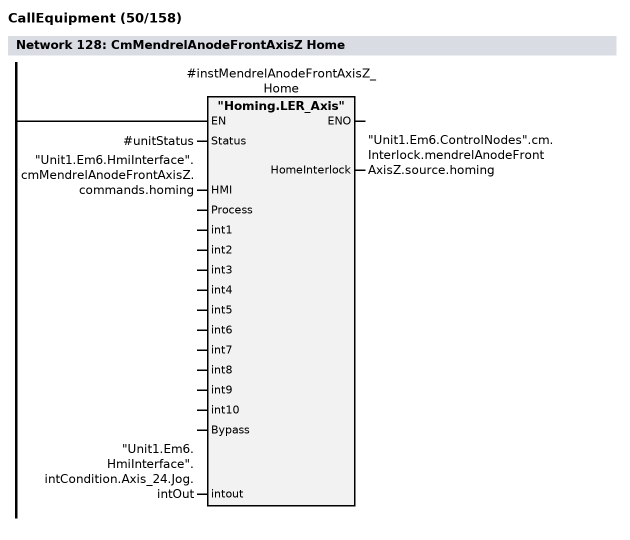
   RUNG wire#powerrail
      #instMendrelAnodeFrontAxisZ_Home(Status := #unitStatus, HMI := "Unit1.Em6.HmiInterface".cmMendrelAnodeFrontAxisZ.commands.homing, Process :=, int1 :=, int2 :=, int3 :=, int4 :=, int5 :=, int6 :=, int7 :=, int8 :=, int9 :=, int10 :=, Bypass :=, intout := "Unit1.Em6.HmiInterface".intCondition.Axis_24.Jog.intOut, HomeInterlock => "Unit1.Em6.ControlNodes".cm.Interlock.mendrelAnodeFrontAxisZ.source.homing)
   END_RUNG
   // the same network as SCL:
   #instMendrelAnodeFrontAxisZ_Home(Status := #unitStatus,   // "Homing.LER_Axis"
                           HMI := "Unit1.Em6.HmiInterface".cmMendrelAnodeFrontAxisZ.commands.homing,
                           intout := "Unit1.Em6.HmiInterface".intCondition.Axis_24.Jog.intOut,
                           HomeInterlock => "Unit1.Em6.ControlNodes".cm.Interlock.mendrelAnodeFrontAxisZ.source.homing);
END_REGION

REGION Network 129: CmmendrelAnodeFrontAxisZ Position Absolute Jog
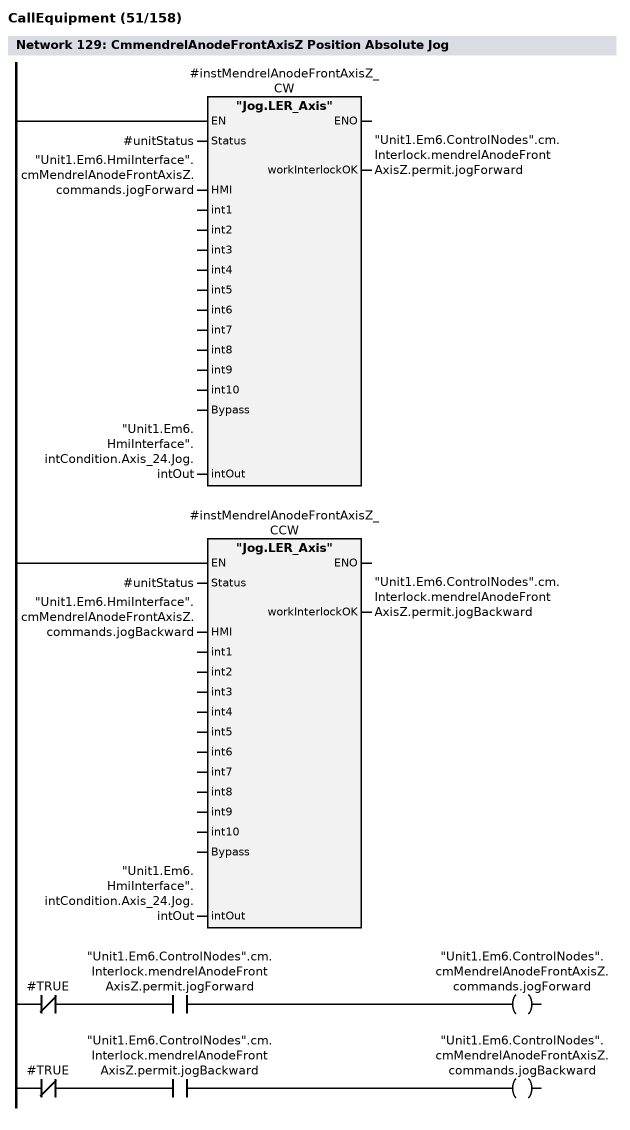
   RUNG wire#powerrail
      #instMendrelAnodeFrontAxisZ_CW(Status := #unitStatus, HMI := "Unit1.Em6.HmiInterface".cmMendrelAnodeFrontAxisZ.commands.jogForward, int1 :=, int2 :=, int3 :=, int4 :=, int5 :=, int6 :=, int7 :=, int8 :=, int9 :=, int10 :=, Bypass :=, intOut := "Unit1.Em6.HmiInterface".intCondition.Axis_24.Jog.intOut, workInterlockOK => "Unit1.Em6.ControlNodes".cm.Interlock.mendrelAnodeFrontAxisZ.permit.jogForward)
   END_RUNG
   RUNG wire#powerrail
      #instMendrelAnodeFrontAxisZ_CCW(Status := #unitStatus, HMI := "Unit1.Em6.HmiInterface".cmMendrelAnodeFrontAxisZ.commands.jogBackward, int1 :=, int2 :=, int3 :=, int4 :=, int5 :=, int6 :=, int7 :=, int8 :=, int9 :=, int10 :=, Bypass :=, intOut := "Unit1.Em6.HmiInterface".intCondition.Axis_24.Jog.intOut, workInterlockOK => "Unit1.Em6.ControlNodes".cm.Interlock.mendrelAnodeFrontAxisZ.permit.jogBackward)
   END_RUNG
   RUNG wire#powerrail
      I_Contact( #TRUE )
      Contact( "Unit1.Em6.ControlNodes".cm.Interlock.mendrelAnodeFrontAxisZ.permit.jogForward )
      Coil( "Unit1.Em6.ControlNodes".cmMendrelAnodeFrontAxisZ.commands.jogForward )
   END_RUNG
   RUNG wire#powerrail
      I_Contact( #TRUE )
      Contact( "Unit1.Em6.ControlNodes".cm.Interlock.mendrelAnodeFrontAxisZ.permit.jogBackward )
      Coil( "Unit1.Em6.ControlNodes".cmMendrelAnodeFrontAxisZ.commands.jogBackward )
   END_RUNG
   // the same network as SCL:
   #instMendrelAnodeFrontAxisZ_CW(Status := #unitStatus,   // "Jog.LER_Axis"
                           HMI := "Unit1.Em6.HmiInterface".cmMendrelAnodeFrontAxisZ.commands.jogForward,
                           intOut := "Unit1.Em6.HmiInterface".intCondition.Axis_24.Jog.intOut,
                           workInterlockOK => "Unit1.Em6.ControlNodes".cm.Interlock.mendrelAnodeFrontAxisZ.permit.jogForward);
   #instMendrelAnodeFrontAxisZ_CCW(Status := #unitStatus,   // "Jog.LER_Axis"
                           HMI := "Unit1.Em6.HmiInterface".cmMendrelAnodeFrontAxisZ.commands.jogBackward,
                           intOut := "Unit1.Em6.HmiInterface".intCondition.Axis_24.Jog.intOut,
                           workInterlockOK => "Unit1.Em6.ControlNodes".cm.Interlock.mendrelAnodeFrontAxisZ.permit.jogBackward);
   "Unit1.Em6.ControlNodes".cmMendrelAnodeFrontAxisZ.commands.jogForward := NOT #TRUE AND "Unit1.Em6.ControlNodes".cm.Interlock.mendrelAnodeFrontAxisZ.permit.jogForward;
   "Unit1.Em6.ControlNodes".cmMendrelAnodeFrontAxisZ.commands.jogBackward := NOT #TRUE AND "Unit1.Em6.ControlNodes".cm.Interlock.mendrelAnodeFrontAxisZ.permit.jogBackward;
END_REGION

REGION Network 130: CmmendrelAnodeFrontAxisZ Position Absolute Position0
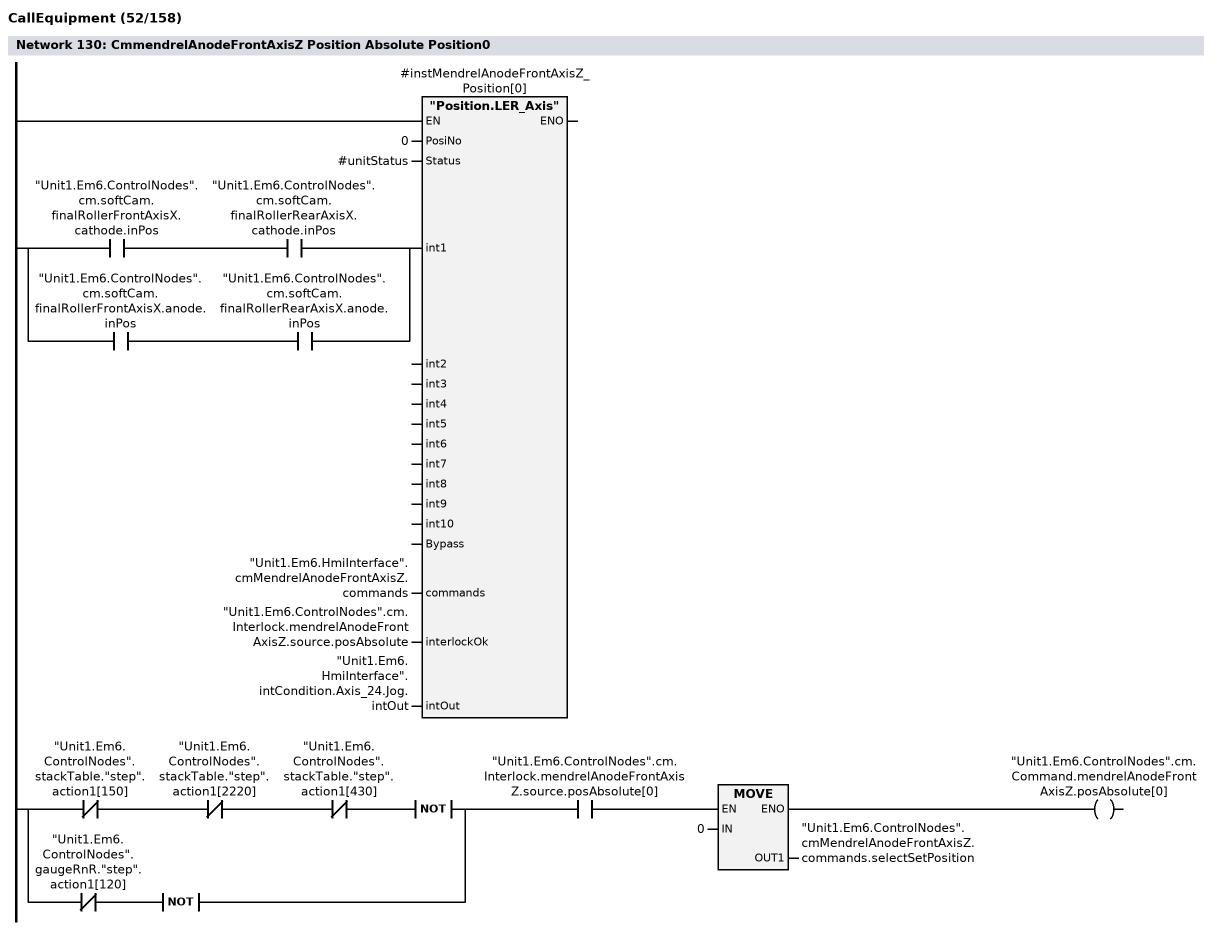
   RUNG wire#powerrail
      #instMendrelAnodeFrontAxisZ_Position[0](int1 := wire#w1, PosiNo := 0, Status := #unitStatus, int2 :=, int3 :=, int4 :=, int5 :=, int6 :=, int7 :=, int8 :=, int9 :=, int10 :=, Bypass :=, commands := "Unit1.Em6.HmiInterface".cmMendrelAnodeFrontAxisZ.commands, interlockOk := "Unit1.Em6.ControlNodes".cm.Interlock.mendrelAnodeFrontAxisZ.source.posAbsolute, intOut := "Unit1.Em6.HmiInterface".intCondition.Axis_24.Jog.intOut)
   END_RUNG
   RUNG wire#powerrail
      Contact( "Unit1.Em6.ControlNodes".cm.softCam.finalRollerFrontAxisX.cathode.inPos )
      Contact( "Unit1.Em6.ControlNodes".cm.softCam.finalRollerRearAxisX.cathode.inPos )
   END_RUNG wire#w1
   RUNG wire#powerrail
      Contact( "Unit1.Em6.ControlNodes".cm.softCam.finalRollerFrontAxisX.anode.inPos )
      Contact( "Unit1.Em6.ControlNodes".cm.softCam.finalRollerRearAxisX.anode.inPos )
   END_RUNG wire#w1
   RUNG wire#powerrail
      I_Contact( "Unit1.Em6.ControlNodes".stackTable."step".action1[150] )
      I_Contact( "Unit1.Em6.ControlNodes".stackTable."step".action1[2220] )
      I_Contact( "Unit1.Em6.ControlNodes".stackTable."step".action1[430] )
      Not()
      wire#w2
      Contact( "Unit1.Em6.ControlNodes".cm.Interlock.mendrelAnodeFrontAxisZ.source.posAbsolute[0] )
      Move(in := 0, out1 => "Unit1.Em6.ControlNodes".cmMendrelAnodeFrontAxisZ.commands.selectSetPosition)
      Coil( "Unit1.Em6.ControlNodes".cm.Command.mendrelAnodeFrontAxisZ.posAbsolute[0] )
   END_RUNG
   RUNG wire#powerrail
      I_Contact( "Unit1.Em6.ControlNodes".gaugeRnR."step".action1[120] )
      Not()
   END_RUNG wire#w2
   // the same network as SCL:
   #instMendrelAnodeFrontAxisZ_Position[0](PosiNo := 0,   // "Position.LER_Axis"
                           Status := #unitStatus,
                           int1 := ("Unit1.Em6.ControlNodes".cm.softCam.finalRollerFrontAxisX.cathode.inPos AND "Unit1.Em6.ControlNodes".cm.softCam.finalRollerRearAxisX.cathode.inPos) OR ("Unit1.Em6.ControlNodes".cm.softCam.finalRollerFrontAxisX.anode.inPos AND "Unit1.Em6.ControlNodes".cm.softCam.finalRollerRearAxisX.anode.inPos),
                           commands := "Unit1.Em6.HmiInterface".cmMendrelAnodeFrontAxisZ.commands,
                           interlockOk := "Unit1.Em6.ControlNodes".cm.Interlock.mendrelAnodeFrontAxisZ.source.posAbsolute,
                           intOut := "Unit1.Em6.HmiInterface".intCondition.Axis_24.Jog.intOut);
   #_w1 := (NOT (NOT "Unit1.Em6.ControlNodes".stackTable."step".action1[150] AND NOT "Unit1.Em6.ControlNodes".stackTable."step".action1[2220] AND NOT "Unit1.Em6.ControlNodes".stackTable."step".action1[430]) OR NOT (NOT "Unit1.Em6.ControlNodes".gaugeRnR."step".action1[120])) AND "Unit1.Em6.ControlNodes".cm.Interlock.mendrelAnodeFrontAxisZ.source.posAbsolute[0];
   IF #_w1 THEN "Unit1.Em6.ControlNodes".cmMendrelAnodeFrontAxisZ.commands.selectSetPosition := 0; END_IF;
   "Unit1.Em6.ControlNodes".cm.Command.mendrelAnodeFrontAxisZ.posAbsolute[0] := #_w1;
END_REGION

REGION Network 131: CmmendrelAnodeFrontAxisZ Position Absolute Position1
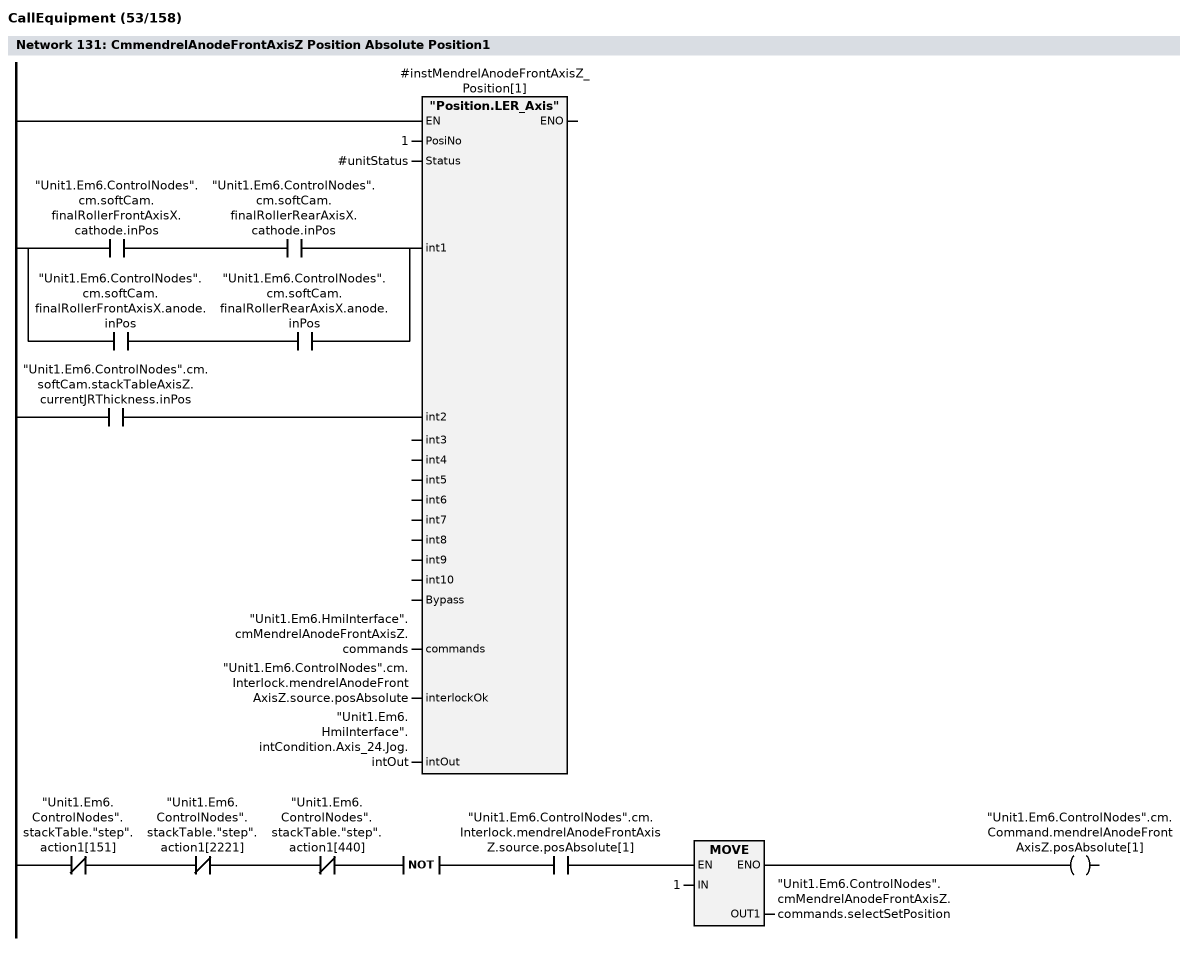
   RUNG wire#powerrail
      #instMendrelAnodeFrontAxisZ_Position[1](int1 := wire#w1, int2 := wire#w2, PosiNo := 1, Status := #unitStatus, int3 :=, int4 :=, int5 :=, int6 :=, int7 :=, int8 :=, int9 :=, int10 :=, Bypass :=, commands := "Unit1.Em6.HmiInterface".cmMendrelAnodeFrontAxisZ.commands, interlockOk := "Unit1.Em6.ControlNodes".cm.Interlock.mendrelAnodeFrontAxisZ.source.posAbsolute, intOut := "Unit1.Em6.HmiInterface".intCondition.Axis_24.Jog.intOut)
   END_RUNG
   RUNG wire#powerrail
      Contact( "Unit1.Em6.ControlNodes".cm.softCam.finalRollerFrontAxisX.cathode.inPos )
      Contact( "Unit1.Em6.ControlNodes".cm.softCam.finalRollerRearAxisX.cathode.inPos )
   END_RUNG wire#w1
   RUNG wire#powerrail
      Contact( "Unit1.Em6.ControlNodes".cm.softCam.finalRollerFrontAxisX.anode.inPos )
      Contact( "Unit1.Em6.ControlNodes".cm.softCam.finalRollerRearAxisX.anode.inPos )
   END_RUNG wire#w1
   RUNG wire#powerrail
      Contact( "Unit1.Em6.ControlNodes".cm.softCam.stackTableAxisZ.currentJRThickness.inPos )
   END_RUNG wire#w2
   RUNG wire#powerrail
      I_Contact( "Unit1.Em6.ControlNodes".stackTable."step".action1[151] )
      I_Contact( "Unit1.Em6.ControlNodes".stackTable."step".action1[2221] )
      I_Contact( "Unit1.Em6.ControlNodes".stackTable."step".action1[440] )
      Not()
      Contact( "Unit1.Em6.ControlNodes".cm.Interlock.mendrelAnodeFrontAxisZ.source.posAbsolute[1] )
      Move(in := 1, out1 => "Unit1.Em6.ControlNodes".cmMendrelAnodeFrontAxisZ.commands.selectSetPosition)
      Coil( "Unit1.Em6.ControlNodes".cm.Command.mendrelAnodeFrontAxisZ.posAbsolute[1] )
   END_RUNG
   // the same network as SCL:
   #instMendrelAnodeFrontAxisZ_Position[1](PosiNo := 1,   // "Position.LER_Axis"
                           Status := #unitStatus,
                           int1 := ("Unit1.Em6.ControlNodes".cm.softCam.finalRollerFrontAxisX.cathode.inPos AND "Unit1.Em6.ControlNodes".cm.softCam.finalRollerRearAxisX.cathode.inPos) OR ("Unit1.Em6.ControlNodes".cm.softCam.finalRollerFrontAxisX.anode.inPos AND "Unit1.Em6.ControlNodes".cm.softCam.finalRollerRearAxisX.anode.inPos),
                           int2 := "Unit1.Em6.ControlNodes".cm.softCam.stackTableAxisZ.currentJRThickness.inPos,
                           commands := "Unit1.Em6.HmiInterface".cmMendrelAnodeFrontAxisZ.commands,
                           interlockOk := "Unit1.Em6.ControlNodes".cm.Interlock.mendrelAnodeFrontAxisZ.source.posAbsolute,
                           intOut := "Unit1.Em6.HmiInterface".intCondition.Axis_24.Jog.intOut);
   #_w1 := NOT (NOT "Unit1.Em6.ControlNodes".stackTable."step".action1[151] AND NOT "Unit1.Em6.ControlNodes".stackTable."step".action1[2221] AND NOT "Unit1.Em6.ControlNodes".stackTable."step".action1[440]) AND "Unit1.Em6.ControlNodes".cm.Interlock.mendrelAnodeFrontAxisZ.source.posAbsolute[1];
   IF #_w1 THEN "Unit1.Em6.ControlNodes".cmMendrelAnodeFrontAxisZ.commands.selectSetPosition := 1; END_IF;
   "Unit1.Em6.ControlNodes".cm.Command.mendrelAnodeFrontAxisZ.posAbsolute[1] := #_w1;
END_REGION

REGION Network 132: CmmendrelAnodeFrontAxisZ Position Absolute Position2
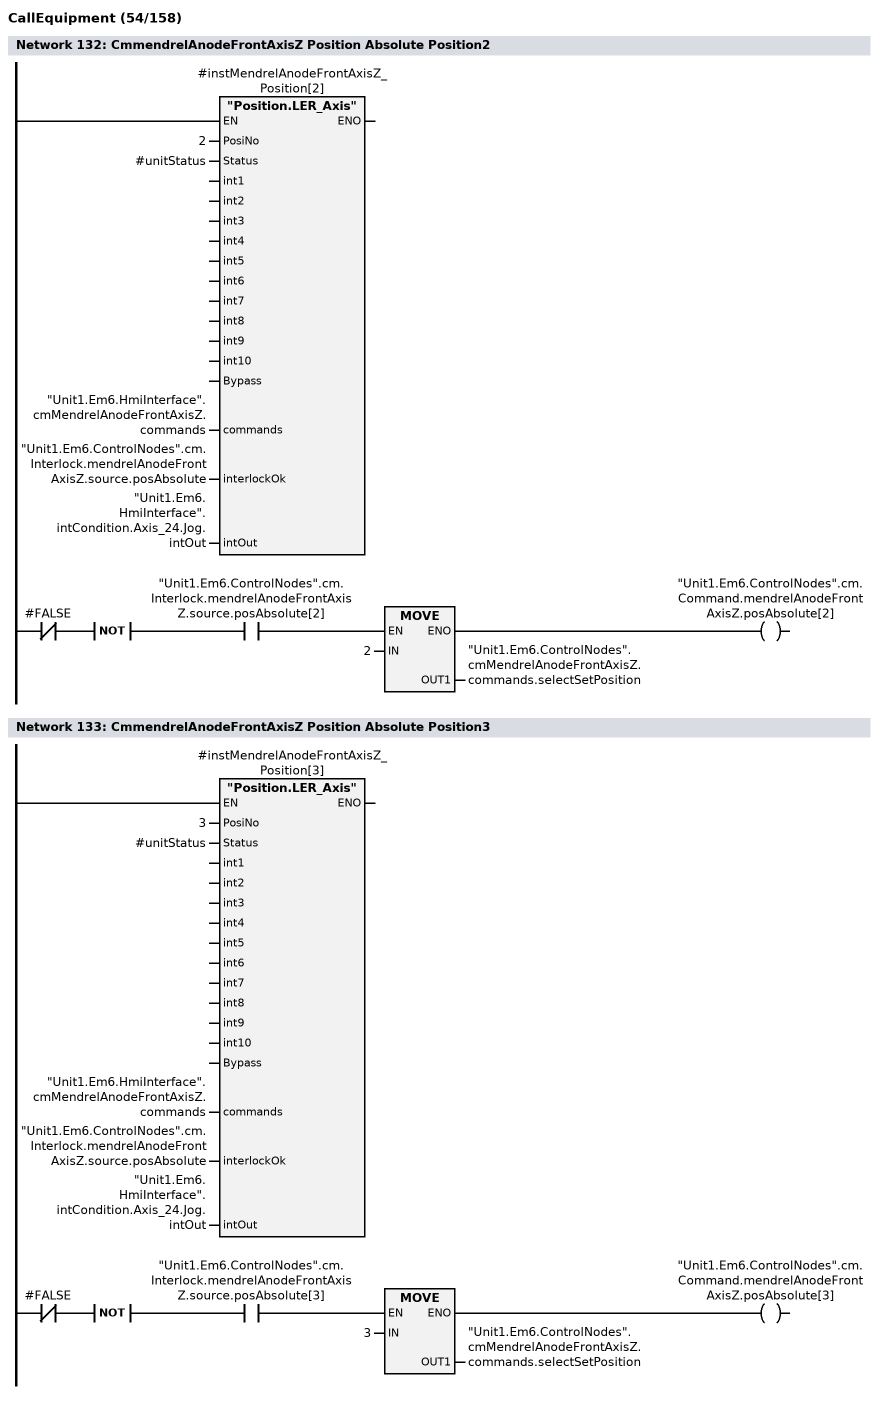
   RUNG wire#powerrail
      #instMendrelAnodeFrontAxisZ_Position[2](PosiNo := 2, Status := #unitStatus, int1 :=, int2 :=, int3 :=, int4 :=, int5 :=, int6 :=, int7 :=, int8 :=, int9 :=, int10 :=, Bypass :=, commands := "Unit1.Em6.HmiInterface".cmMendrelAnodeFrontAxisZ.commands, interlockOk := "Unit1.Em6.ControlNodes".cm.Interlock.mendrelAnodeFrontAxisZ.source.posAbsolute, intOut := "Unit1.Em6.HmiInterface".intCondition.Axis_24.Jog.intOut)
   END_RUNG
   RUNG wire#powerrail
      I_Contact( #FALSE )
      Not()
      Contact( "Unit1.Em6.ControlNodes".cm.Interlock.mendrelAnodeFrontAxisZ.source.posAbsolute[2] )
      Move(in := 2, out1 => "Unit1.Em6.ControlNodes".cmMendrelAnodeFrontAxisZ.commands.selectSetPosition)
      Coil( "Unit1.Em6.ControlNodes".cm.Command.mendrelAnodeFrontAxisZ.posAbsolute[2] )
   END_RUNG
   // the same network as SCL:
   #instMendrelAnodeFrontAxisZ_Position[2](PosiNo := 2,   // "Position.LER_Axis"
                           Status := #unitStatus,
                           commands := "Unit1.Em6.HmiInterface".cmMendrelAnodeFrontAxisZ.commands,
                           interlockOk := "Unit1.Em6.ControlNodes".cm.Interlock.mendrelAnodeFrontAxisZ.source.posAbsolute,
                           intOut := "Unit1.Em6.HmiInterface".intCondition.Axis_24.Jog.intOut);
   #_w1 := NOT (NOT #FALSE) AND "Unit1.Em6.ControlNodes".cm.Interlock.mendrelAnodeFrontAxisZ.source.posAbsolute[2];
   IF #_w1 THEN "Unit1.Em6.ControlNodes".cmMendrelAnodeFrontAxisZ.commands.selectSetPosition := 2; END_IF;
   "Unit1.Em6.ControlNodes".cm.Command.mendrelAnodeFrontAxisZ.posAbsolute[2] := #_w1;
END_REGION

REGION Network 133: CmmendrelAnodeFrontAxisZ Position Absolute Position3
   RUNG wire#powerrail
      #instMendrelAnodeFrontAxisZ_Position[3](PosiNo := 3, Status := #unitStatus, int1 :=, int2 :=, int3 :=, int4 :=, int5 :=, int6 :=, int7 :=, int8 :=, int9 :=, int10 :=, Bypass :=, commands := "Unit1.Em6.HmiInterface".cmMendrelAnodeFrontAxisZ.commands, interlockOk := "Unit1.Em6.ControlNodes".cm.Interlock.mendrelAnodeFrontAxisZ.source.posAbsolute, intOut := "Unit1.Em6.HmiInterface".intCondition.Axis_24.Jog.intOut)
   END_RUNG
   RUNG wire#powerrail
      I_Contact( #FALSE )
      Not()
      Contact( "Unit1.Em6.ControlNodes".cm.Interlock.mendrelAnodeFrontAxisZ.source.posAbsolute[3] )
      Move(in := 3, out1 => "Unit1.Em6.ControlNodes".cmMendrelAnodeFrontAxisZ.commands.selectSetPosition)
      Coil( "Unit1.Em6.ControlNodes".cm.Command.mendrelAnodeFrontAxisZ.posAbsolute[3] )
   END_RUNG
   // the same network as SCL:
   #instMendrelAnodeFrontAxisZ_Position[3](PosiNo := 3,   // "Position.LER_Axis"
                           Status := #unitStatus,
                           commands := "Unit1.Em6.HmiInterface".cmMendrelAnodeFrontAxisZ.commands,
                           interlockOk := "Unit1.Em6.ControlNodes".cm.Interlock.mendrelAnodeFrontAxisZ.source.posAbsolute,
                           intOut := "Unit1.Em6.HmiInterface".intCondition.Axis_24.Jog.intOut);
   #_w1 := NOT (NOT #FALSE) AND "Unit1.Em6.ControlNodes".cm.Interlock.mendrelAnodeFrontAxisZ.source.posAbsolute[3];
   IF #_w1 THEN "Unit1.Em6.ControlNodes".cmMendrelAnodeFrontAxisZ.commands.selectSetPosition := 3; END_IF;
   "Unit1.Em6.ControlNodes".cm.Command.mendrelAnodeFrontAxisZ.posAbsolute[3] := #_w1;
END_REGION

REGION Network 134: CmmendrelAnodeFrontAxisZ Position Absolute Position4
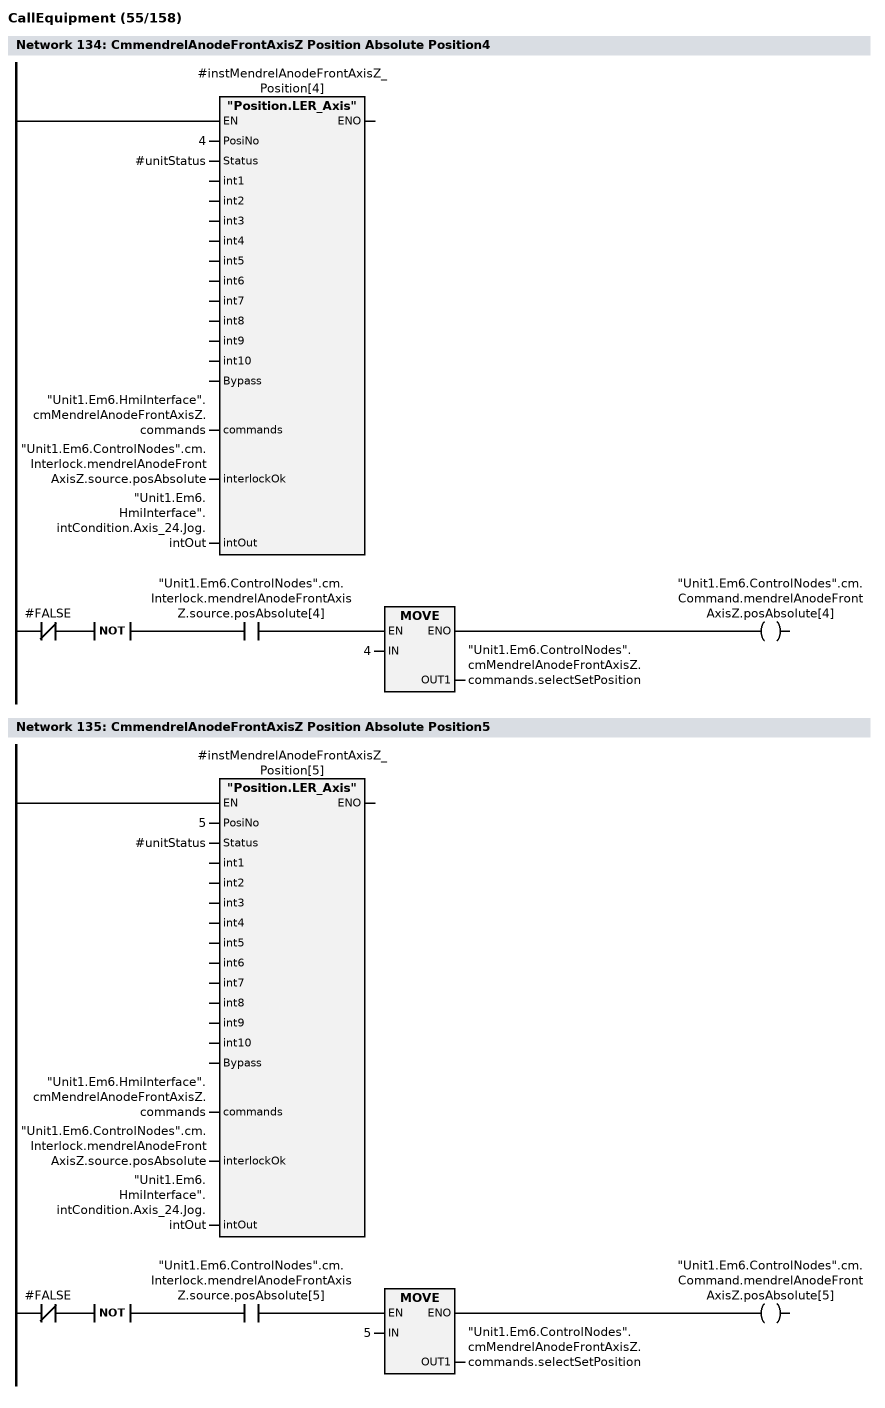
   RUNG wire#powerrail
      #instMendrelAnodeFrontAxisZ_Position[4](PosiNo := 4, Status := #unitStatus, int1 :=, int2 :=, int3 :=, int4 :=, int5 :=, int6 :=, int7 :=, int8 :=, int9 :=, int10 :=, Bypass :=, commands := "Unit1.Em6.HmiInterface".cmMendrelAnodeFrontAxisZ.commands, interlockOk := "Unit1.Em6.ControlNodes".cm.Interlock.mendrelAnodeFrontAxisZ.source.posAbsolute, intOut := "Unit1.Em6.HmiInterface".intCondition.Axis_24.Jog.intOut)
   END_RUNG
   RUNG wire#powerrail
      I_Contact( #FALSE )
      Not()
      Contact( "Unit1.Em6.ControlNodes".cm.Interlock.mendrelAnodeFrontAxisZ.source.posAbsolute[4] )
      Move(in := 4, out1 => "Unit1.Em6.ControlNodes".cmMendrelAnodeFrontAxisZ.commands.selectSetPosition)
      Coil( "Unit1.Em6.ControlNodes".cm.Command.mendrelAnodeFrontAxisZ.posAbsolute[4] )
   END_RUNG
   // the same network as SCL:
   #instMendrelAnodeFrontAxisZ_Position[4](PosiNo := 4,   // "Position.LER_Axis"
                           Status := #unitStatus,
                           commands := "Unit1.Em6.HmiInterface".cmMendrelAnodeFrontAxisZ.commands,
                           interlockOk := "Unit1.Em6.ControlNodes".cm.Interlock.mendrelAnodeFrontAxisZ.source.posAbsolute,
                           intOut := "Unit1.Em6.HmiInterface".intCondition.Axis_24.Jog.intOut);
   #_w1 := NOT (NOT #FALSE) AND "Unit1.Em6.ControlNodes".cm.Interlock.mendrelAnodeFrontAxisZ.source.posAbsolute[4];
   IF #_w1 THEN "Unit1.Em6.ControlNodes".cmMendrelAnodeFrontAxisZ.commands.selectSetPosition := 4; END_IF;
   "Unit1.Em6.ControlNodes".cm.Command.mendrelAnodeFrontAxisZ.posAbsolute[4] := #_w1;
END_REGION

REGION Network 135: CmmendrelAnodeFrontAxisZ Position Absolute Position5
   RUNG wire#powerrail
      #instMendrelAnodeFrontAxisZ_Position[5](PosiNo := 5, Status := #unitStatus, int1 :=, int2 :=, int3 :=, int4 :=, int5 :=, int6 :=, int7 :=, int8 :=, int9 :=, int10 :=, Bypass :=, commands := "Unit1.Em6.HmiInterface".cmMendrelAnodeFrontAxisZ.commands, interlockOk := "Unit1.Em6.ControlNodes".cm.Interlock.mendrelAnodeFrontAxisZ.source.posAbsolute, intOut := "Unit1.Em6.HmiInterface".intCondition.Axis_24.Jog.intOut)
   END_RUNG
   RUNG wire#powerrail
      I_Contact( #FALSE )
      Not()
      Contact( "Unit1.Em6.ControlNodes".cm.Interlock.mendrelAnodeFrontAxisZ.source.posAbsolute[5] )
      Move(in := 5, out1 => "Unit1.Em6.ControlNodes".cmMendrelAnodeFrontAxisZ.commands.selectSetPosition)
      Coil( "Unit1.Em6.ControlNodes".cm.Command.mendrelAnodeFrontAxisZ.posAbsolute[5] )
   END_RUNG
   // the same network as SCL:
   #instMendrelAnodeFrontAxisZ_Position[5](PosiNo := 5,   // "Position.LER_Axis"
                           Status := #unitStatus,
                           commands := "Unit1.Em6.HmiInterface".cmMendrelAnodeFrontAxisZ.commands,
                           interlockOk := "Unit1.Em6.ControlNodes".cm.Interlock.mendrelAnodeFrontAxisZ.source.posAbsolute,
                           intOut := "Unit1.Em6.HmiInterface".intCondition.Axis_24.Jog.intOut);
   #_w1 := NOT (NOT #FALSE) AND "Unit1.Em6.ControlNodes".cm.Interlock.mendrelAnodeFrontAxisZ.source.posAbsolute[5];
   IF #_w1 THEN "Unit1.Em6.ControlNodes".cmMendrelAnodeFrontAxisZ.commands.selectSetPosition := 5; END_IF;
   "Unit1.Em6.ControlNodes".cm.Command.mendrelAnodeFrontAxisZ.posAbsolute[5] := #_w1;
END_REGION

REGION Network 136: CmmendrelAnodeFrontAxisZ Summary Command
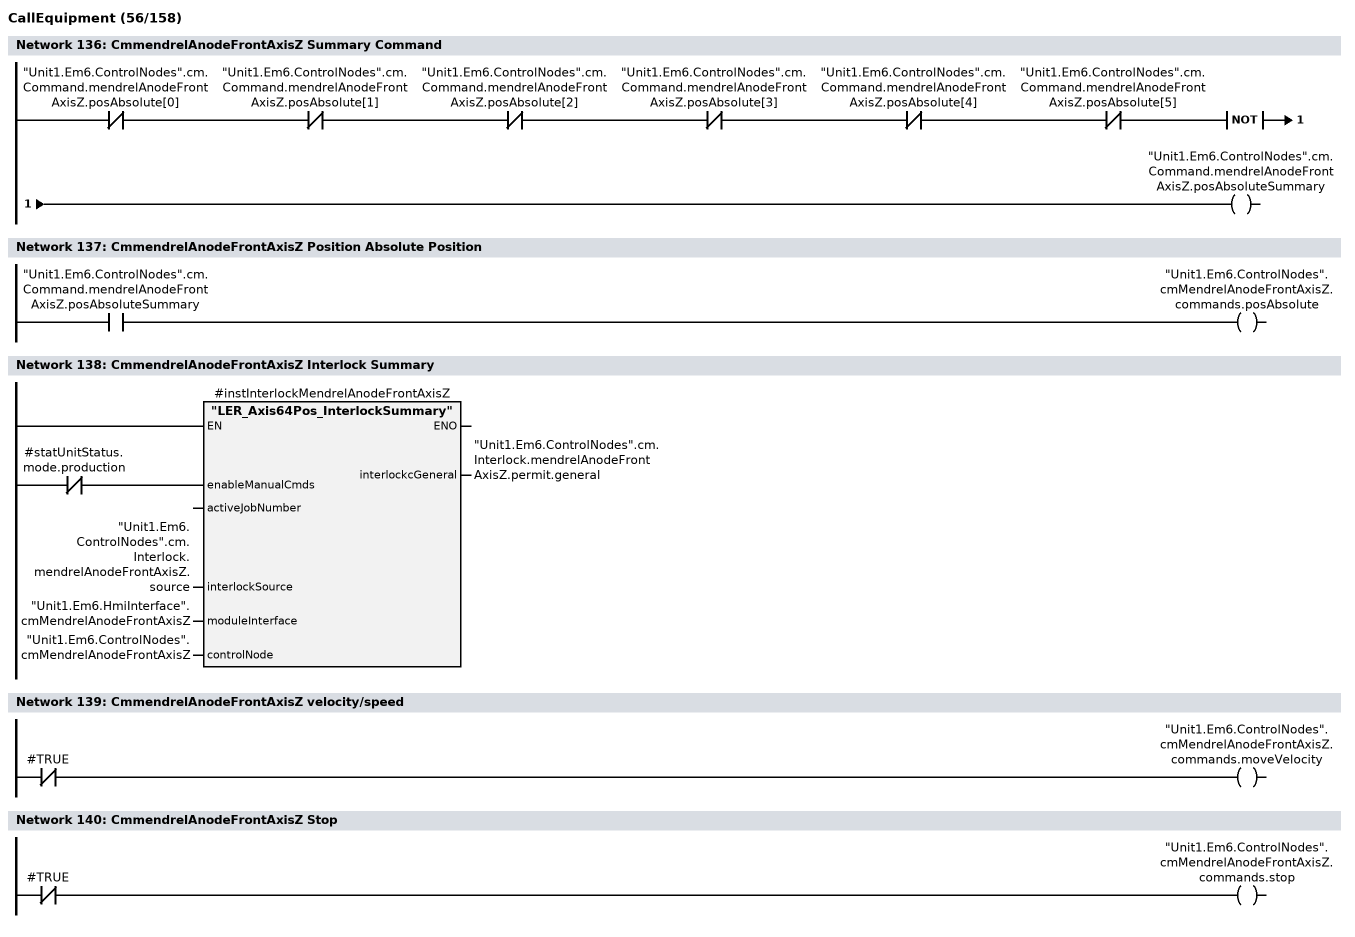
   RUNG wire#powerrail
      I_Contact( "Unit1.Em6.ControlNodes".cm.Command.mendrelAnodeFrontAxisZ.posAbsolute[0] )
      I_Contact( "Unit1.Em6.ControlNodes".cm.Command.mendrelAnodeFrontAxisZ.posAbsolute[1] )
      I_Contact( "Unit1.Em6.ControlNodes".cm.Command.mendrelAnodeFrontAxisZ.posAbsolute[2] )
      I_Contact( "Unit1.Em6.ControlNodes".cm.Command.mendrelAnodeFrontAxisZ.posAbsolute[3] )
      I_Contact( "Unit1.Em6.ControlNodes".cm.Command.mendrelAnodeFrontAxisZ.posAbsolute[4] )
      I_Contact( "Unit1.Em6.ControlNodes".cm.Command.mendrelAnodeFrontAxisZ.posAbsolute[5] )
      Not()
      Coil( "Unit1.Em6.ControlNodes".cm.Command.mendrelAnodeFrontAxisZ.posAbsoluteSummary )
   END_RUNG
   // the same network as SCL:
   "Unit1.Em6.ControlNodes".cm.Command.mendrelAnodeFrontAxisZ.posAbsoluteSummary := NOT (NOT "Unit1.Em6.ControlNodes".cm.Command.mendrelAnodeFrontAxisZ.posAbsolute[0] AND NOT "Unit1.Em6.ControlNodes".cm.Command.mendrelAnodeFrontAxisZ.posAbsolute[1] AND NOT "Unit1.Em6.ControlNodes".cm.Command.mendrelAnodeFrontAxisZ.posAbsolute[2] AND NOT "Unit1.Em6.ControlNodes".cm.Command.mendrelAnodeFrontAxisZ.posAbsolute[3] AND NOT "Unit1.Em6.ControlNodes".cm.Command.mendrelAnodeFrontAxisZ.posAbsolute[4] AND NOT "Unit1.Em6.ControlNodes".cm.Command.mendrelAnodeFrontAxisZ.posAbsolute[5]);
END_REGION

REGION Network 137: CmmendrelAnodeFrontAxisZ Position Absolute Position
   RUNG wire#powerrail
      Contact( "Unit1.Em6.ControlNodes".cm.Command.mendrelAnodeFrontAxisZ.posAbsoluteSummary )
      Coil( "Unit1.Em6.ControlNodes".cmMendrelAnodeFrontAxisZ.commands.posAbsolute )
   END_RUNG
   // the same network as SCL:
   "Unit1.Em6.ControlNodes".cmMendrelAnodeFrontAxisZ.commands.posAbsolute := "Unit1.Em6.ControlNodes".cm.Command.mendrelAnodeFrontAxisZ.posAbsoluteSummary;
END_REGION

REGION Network 138: CmmendrelAnodeFrontAxisZ Interlock Summary
   RUNG wire#powerrail
      #instInterlockMendrelAnodeFrontAxisZ(enableManualCmds := wire#w1, activeJobNumber :=, interlockSource := "Unit1.Em6.ControlNodes".cm.Interlock.mendrelAnodeFrontAxisZ.source, moduleInterface := "Unit1.Em6.HmiInterface".cmMendrelAnodeFrontAxisZ, controlNode := "Unit1.Em6.ControlNodes".cmMendrelAnodeFrontAxisZ, interlockcGeneral => "Unit1.Em6.ControlNodes".cm.Interlock.mendrelAnodeFrontAxisZ.permit.general)
   END_RUNG
   RUNG wire#powerrail
      I_Contact( #statUnitStatus.mode.production )
   END_RUNG wire#w1
   // the same network as SCL:
   #instInterlockMendrelAnodeFrontAxisZ(enableManualCmds := NOT #statUnitStatus.mode.production,   // "LER_Axis64Pos_InterlockSummary"
                           interlockSource := "Unit1.Em6.ControlNodes".cm.Interlock.mendrelAnodeFrontAxisZ.source,
                           moduleInterface := "Unit1.Em6.HmiInterface".cmMendrelAnodeFrontAxisZ,
                           controlNode := "Unit1.Em6.ControlNodes".cmMendrelAnodeFrontAxisZ,
                           interlockcGeneral => "Unit1.Em6.ControlNodes".cm.Interlock.mendrelAnodeFrontAxisZ.permit.general);
END_REGION

REGION Network 139: CmmendrelAnodeFrontAxisZ velocity/speed
   RUNG wire#powerrail
      I_Contact( #TRUE )
      Coil( "Unit1.Em6.ControlNodes".cmMendrelAnodeFrontAxisZ.commands.moveVelocity )
   END_RUNG
   // the same network as SCL:
   "Unit1.Em6.ControlNodes".cmMendrelAnodeFrontAxisZ.commands.moveVelocity := NOT #TRUE;
END_REGION

REGION Network 140: CmmendrelAnodeFrontAxisZ Stop
   RUNG wire#powerrail
      I_Contact( #TRUE )
      Coil( "Unit1.Em6.ControlNodes".cmMendrelAnodeFrontAxisZ.commands.stop )
   END_RUNG
   // the same network as SCL:
   "Unit1.Em6.ControlNodes".cmMendrelAnodeFrontAxisZ.commands.stop := NOT #TRUE;
END_REGION

REGION Network 141: Call CM Anode Mandrel Front Z-Axis (LBC_Axis64Pos)
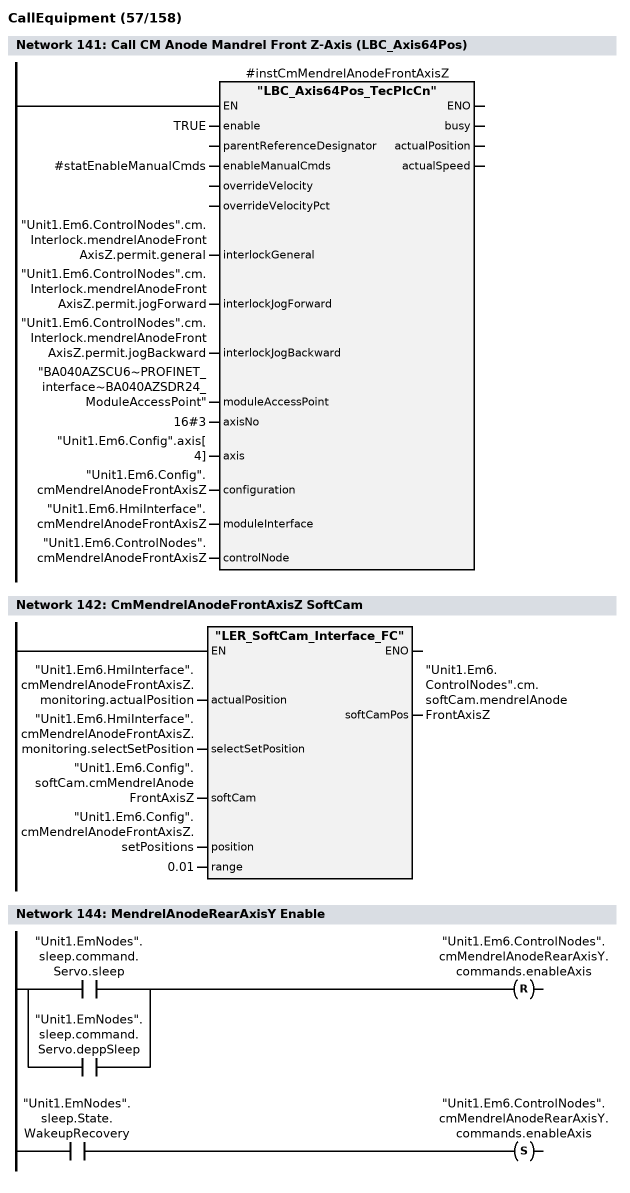
   RUNG wire#powerrail
      #instCmMendrelAnodeFrontAxisZ(enable := TRUE, parentReferenceDesignator :=, enableManualCmds := #statEnableManualCmds, overrideVelocity :=, overrideVelocityPct :=, interlockGeneral := "Unit1.Em6.ControlNodes".cm.Interlock.mendrelAnodeFrontAxisZ.permit.general, interlockJogForward := "Unit1.Em6.ControlNodes".cm.Interlock.mendrelAnodeFrontAxisZ.permit.jogForward, interlockJogBackward := "Unit1.Em6.ControlNodes".cm.Interlock.mendrelAnodeFrontAxisZ.permit.jogBackward, moduleAccessPoint := "BA040AZSCU6~PROFINET_interface~BA040AZSDR24_ModuleAccessPoint", axisNo := 16#3, axis := "Unit1.Em6.Config".axis[4], configuration := "Unit1.Em6.Config".cmMendrelAnodeFrontAxisZ, moduleInterface := "Unit1.Em6.HmiInterface".cmMendrelAnodeFrontAxisZ, controlNode := "Unit1.Em6.ControlNodes".cmMendrelAnodeFrontAxisZ, busy =>, actualPosition =>, actualSpeed =>)
   END_RUNG
   // the same network as SCL:
   #instCmMendrelAnodeFrontAxisZ(enable := TRUE,   // "LBC_Axis64Pos_TecPlcCn"
                           enableManualCmds := #statEnableManualCmds,
                           interlockGeneral := "Unit1.Em6.ControlNodes".cm.Interlock.mendrelAnodeFrontAxisZ.permit.general,
                           interlockJogForward := "Unit1.Em6.ControlNodes".cm.Interlock.mendrelAnodeFrontAxisZ.permit.jogForward,
                           interlockJogBackward := "Unit1.Em6.ControlNodes".cm.Interlock.mendrelAnodeFrontAxisZ.permit.jogBackward,
                           moduleAccessPoint := "BA040AZSCU6~PROFINET_interface~BA040AZSDR24_ModuleAccessPoint",
                           axisNo := 16#3,
                           axis := "Unit1.Em6.Config".axis[4],
                           configuration := "Unit1.Em6.Config".cmMendrelAnodeFrontAxisZ,
                           moduleInterface := "Unit1.Em6.HmiInterface".cmMendrelAnodeFrontAxisZ,
                           controlNode := "Unit1.Em6.ControlNodes".cmMendrelAnodeFrontAxisZ);
END_REGION

REGION Network 142: CmMendrelAnodeFrontAxisZ SoftCam
   RUNG wire#powerrail
      "LER_SoftCam_Interface_FC"(actualPosition := "Unit1.Em6.HmiInterface".cmMendrelAnodeFrontAxisZ.monitoring.actualPosition, selectSetPosition := "Unit1.Em6.HmiInterface".cmMendrelAnodeFrontAxisZ.monitoring.selectSetPosition, softCam := "Unit1.Em6.Config".softCam.cmMendrelAnodeFrontAxisZ, position := "Unit1.Em6.Config".cmMendrelAnodeFrontAxisZ.setPositions, range := 0.01, softCamPos => "Unit1.Em6.ControlNodes".cm.softCam.mendrelAnodeFrontAxisZ)
   END_RUNG
   // the same network as SCL:
   "LER_SoftCam_Interface_FC"(actualPosition := "Unit1.Em6.HmiInterface".cmMendrelAnodeFrontAxisZ.monitoring.actualPosition,
                           selectSetPosition := "Unit1.Em6.HmiInterface".cmMendrelAnodeFrontAxisZ.monitoring.selectSetPosition,
                           softCam := "Unit1.Em6.Config".softCam.cmMendrelAnodeFrontAxisZ,
                           position := "Unit1.Em6.Config".cmMendrelAnodeFrontAxisZ.setPositions,
                           range := 0.01,
                           softCamPos => "Unit1.Em6.ControlNodes".cm.softCam.mendrelAnodeFrontAxisZ);
END_REGION

REGION Network 144: MendrelAnodeRearAxisY Enable
   RUNG wire#powerrail
      Contact( "Unit1.EmNodes".sleep.command.Servo.sleep )
      wire#w1
      R_Coil( "Unit1.Em6.ControlNodes".cmMendrelAnodeRearAxisY.commands.enableAxis )
   END_RUNG
   RUNG wire#powerrail
      Contact( "Unit1.EmNodes".sleep.command.Servo.deppSleep )
   END_RUNG wire#w1
   RUNG wire#powerrail
      Contact( "Unit1.EmNodes".sleep.State.WakeupRecovery )
      S_Coil( "Unit1.Em6.ControlNodes".cmMendrelAnodeRearAxisY.commands.enableAxis )
   END_RUNG
   // the same network as SCL:
   IF "Unit1.EmNodes".sleep.command.Servo.sleep OR "Unit1.EmNodes".sleep.command.Servo.deppSleep THEN
       "Unit1.Em6.ControlNodes".cmMendrelAnodeRearAxisY.commands.enableAxis := FALSE;
   END_IF;
   IF "Unit1.EmNodes".sleep.State.WakeupRecovery THEN
       "Unit1.Em6.ControlNodes".cmMendrelAnodeRearAxisY.commands.enableAxis := TRUE;
   END_IF;
END_REGION

REGION Network 145: CmMandrelAnodeRearAxisY Home
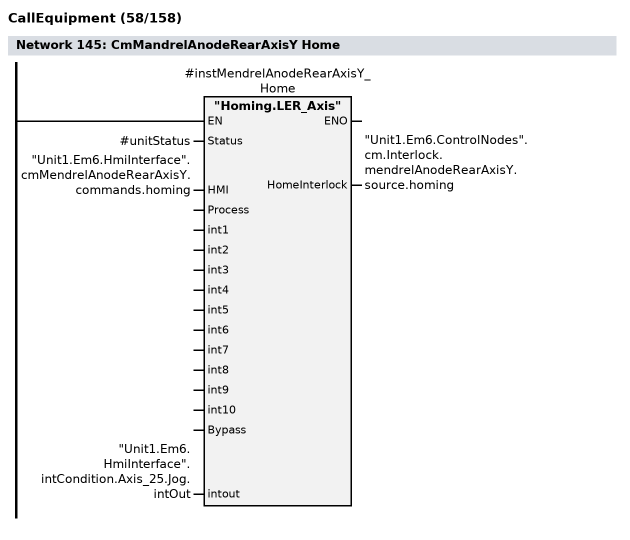
   RUNG wire#powerrail
      #instMendrelAnodeRearAxisY_Home(Status := #unitStatus, HMI := "Unit1.Em6.HmiInterface".cmMendrelAnodeRearAxisY.commands.homing, Process :=, int1 :=, int2 :=, int3 :=, int4 :=, int5 :=, int6 :=, int7 :=, int8 :=, int9 :=, int10 :=, Bypass :=, intout := "Unit1.Em6.HmiInterface".intCondition.Axis_25.Jog.intOut, HomeInterlock => "Unit1.Em6.ControlNodes".cm.Interlock.mendrelAnodeRearAxisY.source.homing)
   END_RUNG
   // the same network as SCL:
   #instMendrelAnodeRearAxisY_Home(Status := #unitStatus,   // "Homing.LER_Axis"
                           HMI := "Unit1.Em6.HmiInterface".cmMendrelAnodeRearAxisY.commands.homing,
                           intout := "Unit1.Em6.HmiInterface".intCondition.Axis_25.Jog.intOut,
                           HomeInterlock => "Unit1.Em6.ControlNodes".cm.Interlock.mendrelAnodeRearAxisY.source.homing);
END_REGION

REGION Network 146: CmMendrelAnodeRearAxisY Position Absolute Jog
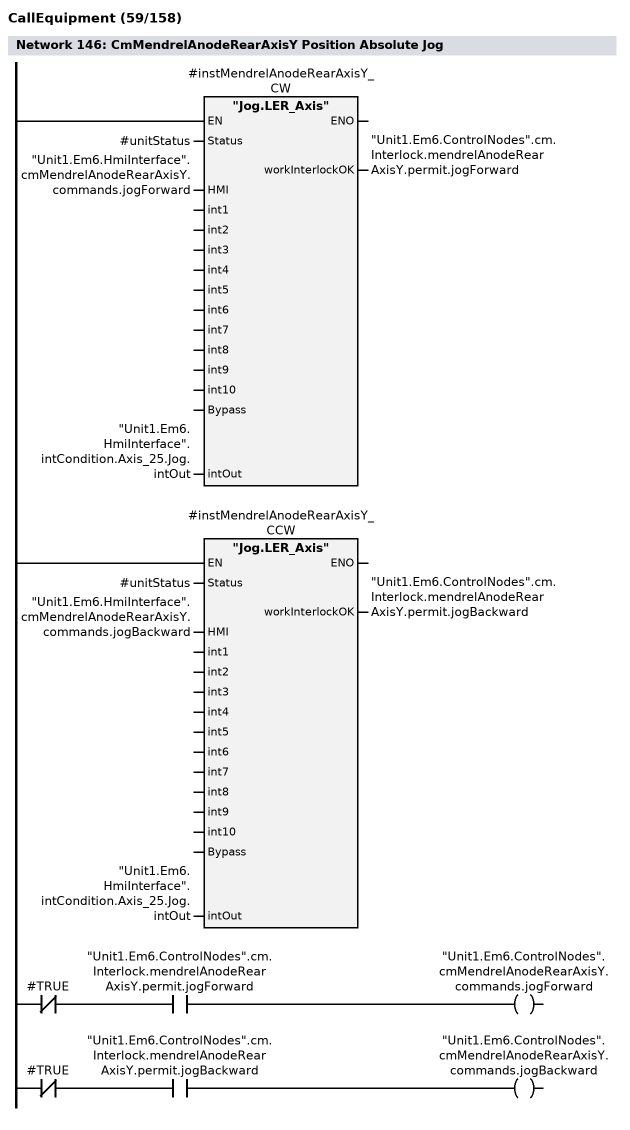
   RUNG wire#powerrail
      #instMendrelAnodeRearAxisY_CW(Status := #unitStatus, HMI := "Unit1.Em6.HmiInterface".cmMendrelAnodeRearAxisY.commands.jogForward, int1 :=, int2 :=, int3 :=, int4 :=, int5 :=, int6 :=, int7 :=, int8 :=, int9 :=, int10 :=, Bypass :=, intOut := "Unit1.Em6.HmiInterface".intCondition.Axis_25.Jog.intOut, workInterlockOK => "Unit1.Em6.ControlNodes".cm.Interlock.mendrelAnodeRearAxisY.permit.jogForward)
   END_RUNG
   RUNG wire#powerrail
      #instMendrelAnodeRearAxisY_CCW(Status := #unitStatus, HMI := "Unit1.Em6.HmiInterface".cmMendrelAnodeRearAxisY.commands.jogBackward, int1 :=, int2 :=, int3 :=, int4 :=, int5 :=, int6 :=, int7 :=, int8 :=, int9 :=, int10 :=, Bypass :=, intOut := "Unit1.Em6.HmiInterface".intCondition.Axis_25.Jog.intOut, workInterlockOK => "Unit1.Em6.ControlNodes".cm.Interlock.mendrelAnodeRearAxisY.permit.jogBackward)
   END_RUNG
   RUNG wire#powerrail
      I_Contact( #TRUE )
      Contact( "Unit1.Em6.ControlNodes".cm.Interlock.mendrelAnodeRearAxisY.permit.jogForward )
      Coil( "Unit1.Em6.ControlNodes".cmMendrelAnodeRearAxisY.commands.jogForward )
   END_RUNG
   RUNG wire#powerrail
      I_Contact( #TRUE )
      Contact( "Unit1.Em6.ControlNodes".cm.Interlock.mendrelAnodeRearAxisY.permit.jogBackward )
      Coil( "Unit1.Em6.ControlNodes".cmMendrelAnodeRearAxisY.commands.jogBackward )
   END_RUNG
   // the same network as SCL:
   #instMendrelAnodeRearAxisY_CW(Status := #unitStatus,   // "Jog.LER_Axis"
                           HMI := "Unit1.Em6.HmiInterface".cmMendrelAnodeRearAxisY.commands.jogForward,
                           intOut := "Unit1.Em6.HmiInterface".intCondition.Axis_25.Jog.intOut,
                           workInterlockOK => "Unit1.Em6.ControlNodes".cm.Interlock.mendrelAnodeRearAxisY.permit.jogForward);
   #instMendrelAnodeRearAxisY_CCW(Status := #unitStatus,   // "Jog.LER_Axis"
                           HMI := "Unit1.Em6.HmiInterface".cmMendrelAnodeRearAxisY.commands.jogBackward,
                           intOut := "Unit1.Em6.HmiInterface".intCondition.Axis_25.Jog.intOut,
                           workInterlockOK => "Unit1.Em6.ControlNodes".cm.Interlock.mendrelAnodeRearAxisY.permit.jogBackward);
   "Unit1.Em6.ControlNodes".cmMendrelAnodeRearAxisY.commands.jogForward := NOT #TRUE AND "Unit1.Em6.ControlNodes".cm.Interlock.mendrelAnodeRearAxisY.permit.jogForward;
   "Unit1.Em6.ControlNodes".cmMendrelAnodeRearAxisY.commands.jogBackward := NOT #TRUE AND "Unit1.Em6.ControlNodes".cm.Interlock.mendrelAnodeRearAxisY.permit.jogBackward;
END_REGION

REGION Network 147: CmMendrelAnodeRearAxisY Position Absolute Position0
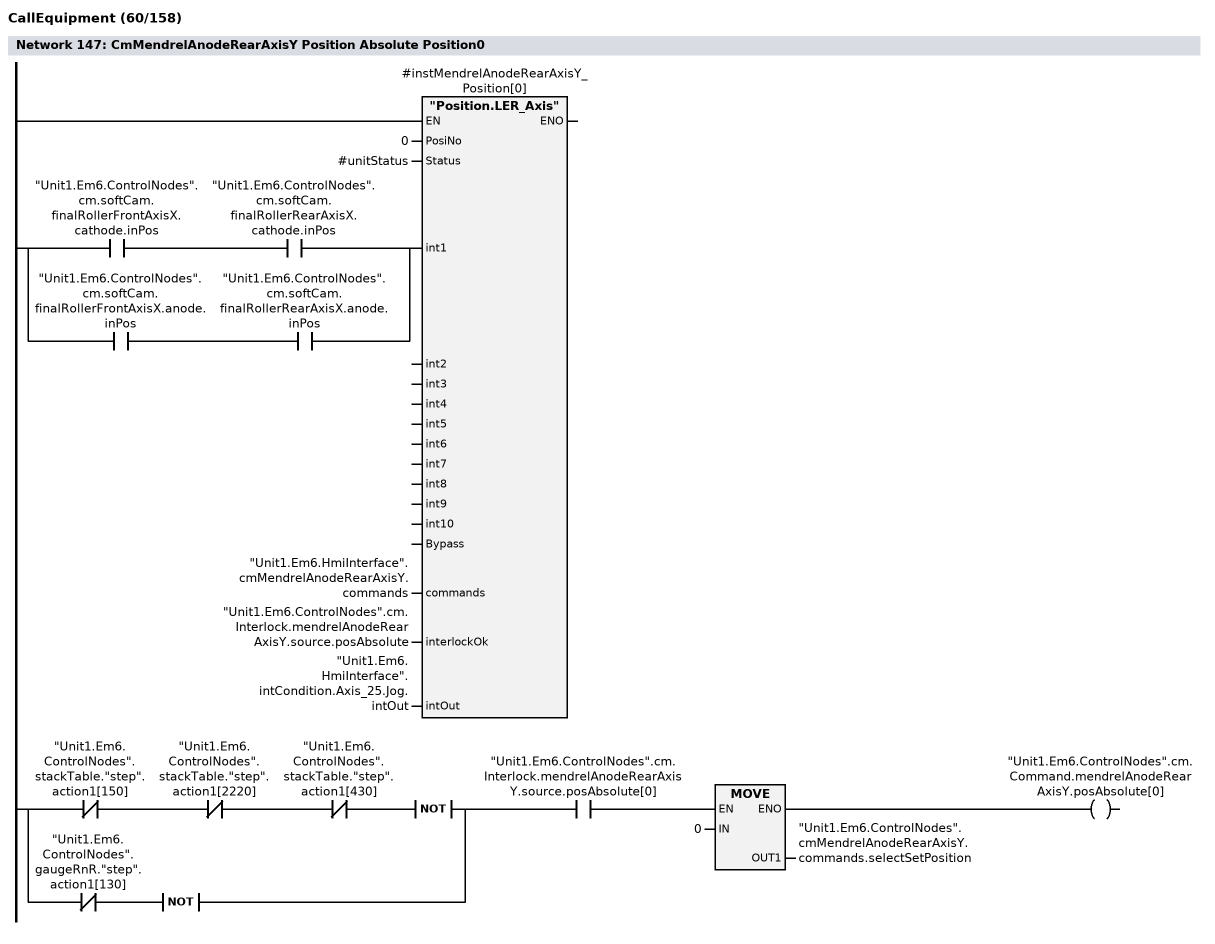
   RUNG wire#powerrail
      #instMendrelAnodeRearAxisY_Position[0](int1 := wire#w1, PosiNo := 0, Status := #unitStatus, int2 :=, int3 :=, int4 :=, int5 :=, int6 :=, int7 :=, int8 :=, int9 :=, int10 :=, Bypass :=, commands := "Unit1.Em6.HmiInterface".cmMendrelAnodeRearAxisY.commands, interlockOk := "Unit1.Em6.ControlNodes".cm.Interlock.mendrelAnodeRearAxisY.source.posAbsolute, intOut := "Unit1.Em6.HmiInterface".intCondition.Axis_25.Jog.intOut)
   END_RUNG
   RUNG wire#powerrail
      Contact( "Unit1.Em6.ControlNodes".cm.softCam.finalRollerFrontAxisX.cathode.inPos )
      Contact( "Unit1.Em6.ControlNodes".cm.softCam.finalRollerRearAxisX.cathode.inPos )
   END_RUNG wire#w1
   RUNG wire#powerrail
      Contact( "Unit1.Em6.ControlNodes".cm.softCam.finalRollerFrontAxisX.anode.inPos )
      Contact( "Unit1.Em6.ControlNodes".cm.softCam.finalRollerRearAxisX.anode.inPos )
   END_RUNG wire#w1
   RUNG wire#powerrail
      I_Contact( "Unit1.Em6.ControlNodes".stackTable."step".action1[150] )
      I_Contact( "Unit1.Em6.ControlNodes".stackTable."step".action1[2220] )
      I_Contact( "Unit1.Em6.ControlNodes".stackTable."step".action1[430] )
      Not()
      wire#w2
      Contact( "Unit1.Em6.ControlNodes".cm.Interlock.mendrelAnodeRearAxisY.source.posAbsolute[0] )
      Move(in := 0, out1 => "Unit1.Em6.ControlNodes".cmMendrelAnodeRearAxisY.commands.selectSetPosition)
      Coil( "Unit1.Em6.ControlNodes".cm.Command.mendrelAnodeRearAxisY.posAbsolute[0] )
   END_RUNG
   RUNG wire#powerrail
      I_Contact( "Unit1.Em6.ControlNodes".gaugeRnR."step".action1[130] )
      Not()
   END_RUNG wire#w2
   // the same network as SCL:
   #instMendrelAnodeRearAxisY_Position[0](PosiNo := 0,   // "Position.LER_Axis"
                           Status := #unitStatus,
                           int1 := ("Unit1.Em6.ControlNodes".cm.softCam.finalRollerFrontAxisX.cathode.inPos AND "Unit1.Em6.ControlNodes".cm.softCam.finalRollerRearAxisX.cathode.inPos) OR ("Unit1.Em6.ControlNodes".cm.softCam.finalRollerFrontAxisX.anode.inPos AND "Unit1.Em6.ControlNodes".cm.softCam.finalRollerRearAxisX.anode.inPos),
                           commands := "Unit1.Em6.HmiInterface".cmMendrelAnodeRearAxisY.commands,
                           interlockOk := "Unit1.Em6.ControlNodes".cm.Interlock.mendrelAnodeRearAxisY.source.posAbsolute,
                           intOut := "Unit1.Em6.HmiInterface".intCondition.Axis_25.Jog.intOut);
   #_w1 := (NOT (NOT "Unit1.Em6.ControlNodes".stackTable."step".action1[150] AND NOT "Unit1.Em6.ControlNodes".stackTable."step".action1[2220] AND NOT "Unit1.Em6.ControlNodes".stackTable."step".action1[430]) OR NOT (NOT "Unit1.Em6.ControlNodes".gaugeRnR."step".action1[130])) AND "Unit1.Em6.ControlNodes".cm.Interlock.mendrelAnodeRearAxisY.source.posAbsolute[0];
   IF #_w1 THEN "Unit1.Em6.ControlNodes".cmMendrelAnodeRearAxisY.commands.selectSetPosition := 0; END_IF;
   "Unit1.Em6.ControlNodes".cm.Command.mendrelAnodeRearAxisY.posAbsolute[0] := #_w1;
END_REGION

REGION Network 148: CmMendrelAnodeRearAxisY Position Absolute Position1
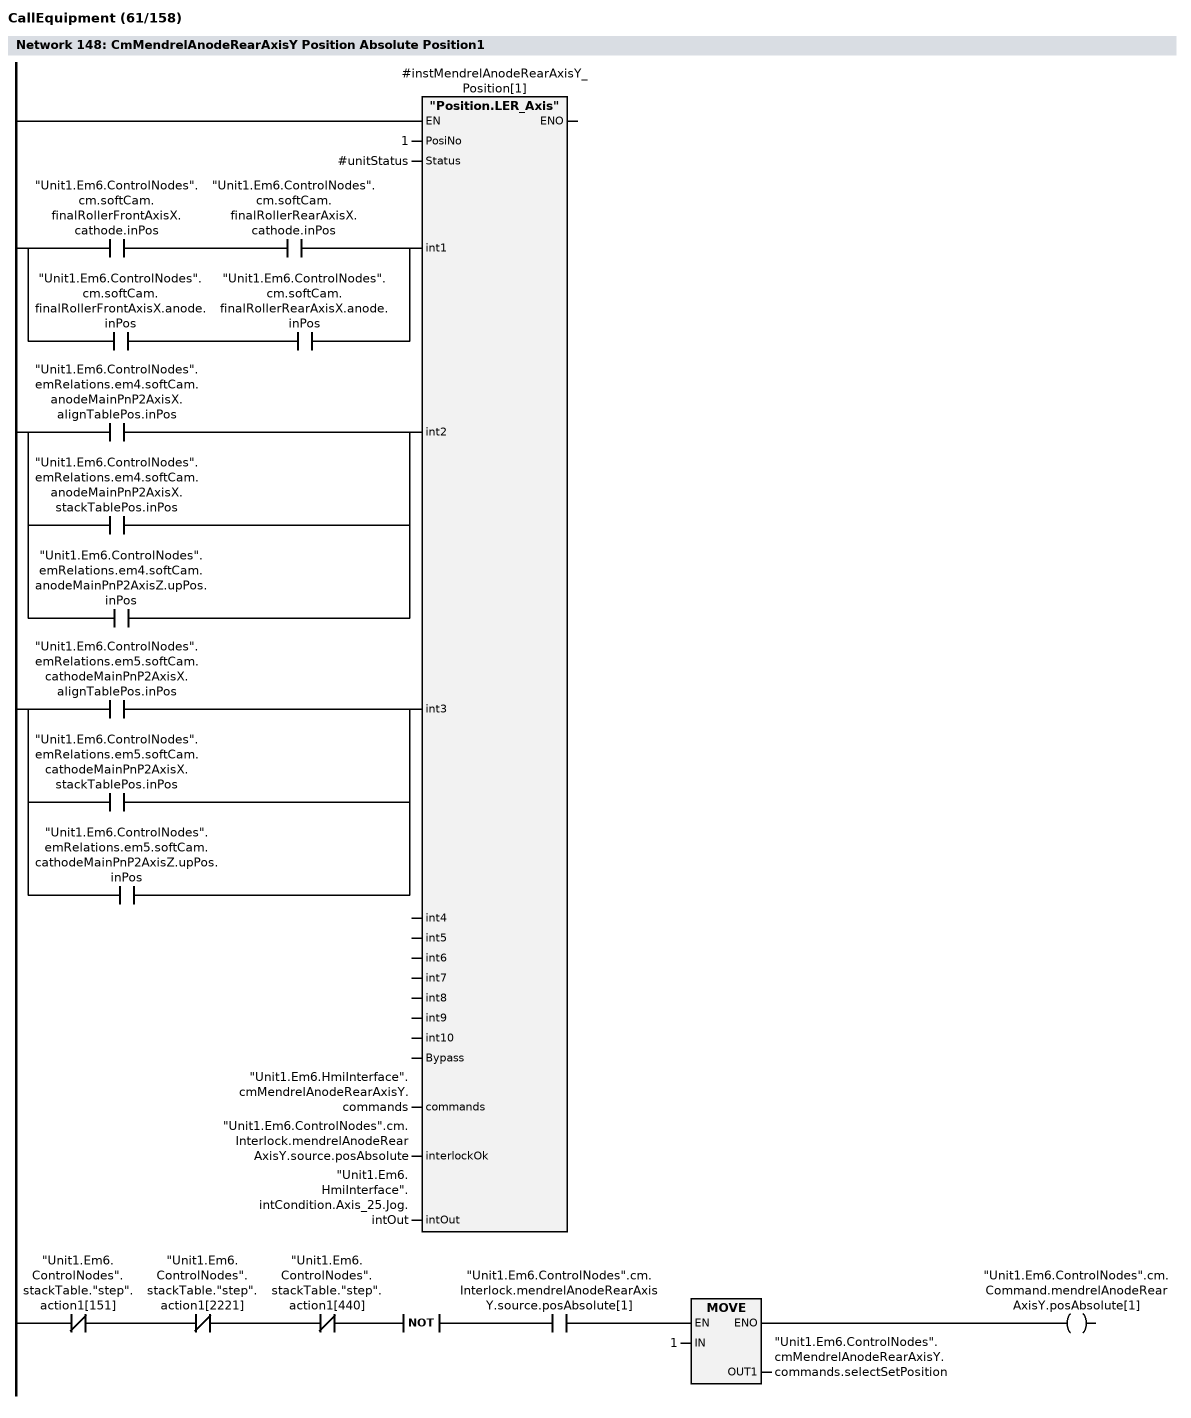
   RUNG wire#powerrail
      #instMendrelAnodeRearAxisY_Position[1](int1 := wire#w1, int2 := wire#w2, int3 := wire#w3, PosiNo := 1, Status := #unitStatus, int4 :=, int5 :=, int6 :=, int7 :=, int8 :=, int9 :=, int10 :=, Bypass :=, commands := "Unit1.Em6.HmiInterface".cmMendrelAnodeRearAxisY.commands, interlockOk := "Unit1.Em6.ControlNodes".cm.Interlock.mendrelAnodeRearAxisY.source.posAbsolute, intOut := "Unit1.Em6.HmiInterface".intCondition.Axis_25.Jog.intOut)
   END_RUNG
   RUNG wire#powerrail
      Contact( "Unit1.Em6.ControlNodes".cm.softCam.finalRollerFrontAxisX.cathode.inPos )
      Contact( "Unit1.Em6.ControlNodes".cm.softCam.finalRollerRearAxisX.cathode.inPos )
   END_RUNG wire#w1
   RUNG wire#powerrail
      Contact( "Unit1.Em6.ControlNodes".cm.softCam.finalRollerFrontAxisX.anode.inPos )
      Contact( "Unit1.Em6.ControlNodes".cm.softCam.finalRollerRearAxisX.anode.inPos )
   END_RUNG wire#w1
   RUNG wire#powerrail
      Contact( "Unit1.Em6.ControlNodes".emRelations.em4.softCam.anodeMainPnP2AxisX.alignTablePos.inPos )
   END_RUNG wire#w2
   RUNG wire#powerrail
      Contact( "Unit1.Em6.ControlNodes".emRelations.em4.softCam.anodeMainPnP2AxisX.stackTablePos.inPos )
   END_RUNG wire#w2
   RUNG wire#powerrail
      Contact( "Unit1.Em6.ControlNodes".emRelations.em4.softCam.anodeMainPnP2AxisZ.upPos.inPos )
   END_RUNG wire#w2
   RUNG wire#powerrail
      Contact( "Unit1.Em6.ControlNodes".emRelations.em5.softCam.cathodeMainPnP2AxisX.alignTablePos.inPos )
   END_RUNG wire#w3
   RUNG wire#powerrail
      Contact( "Unit1.Em6.ControlNodes".emRelations.em5.softCam.cathodeMainPnP2AxisX.stackTablePos.inPos )
   END_RUNG wire#w3
   RUNG wire#powerrail
      Contact( "Unit1.Em6.ControlNodes".emRelations.em5.softCam.cathodeMainPnP2AxisZ.upPos.inPos )
   END_RUNG wire#w3
   RUNG wire#powerrail
      I_Contact( "Unit1.Em6.ControlNodes".stackTable."step".action1[151] )
      I_Contact( "Unit1.Em6.ControlNodes".stackTable."step".action1[2221] )
      I_Contact( "Unit1.Em6.ControlNodes".stackTable."step".action1[440] )
      Not()
      Contact( "Unit1.Em6.ControlNodes".cm.Interlock.mendrelAnodeRearAxisY.source.posAbsolute[1] )
      Move(in := 1, out1 => "Unit1.Em6.ControlNodes".cmMendrelAnodeRearAxisY.commands.selectSetPosition)
      Coil( "Unit1.Em6.ControlNodes".cm.Command.mendrelAnodeRearAxisY.posAbsolute[1] )
   END_RUNG
   // the same network as SCL:
   #instMendrelAnodeRearAxisY_Position[1](PosiNo := 1,   // "Position.LER_Axis"
                           Status := #unitStatus,
                           int1 := ("Unit1.Em6.ControlNodes".cm.softCam.finalRollerFrontAxisX.cathode.inPos AND "Unit1.Em6.ControlNodes".cm.softCam.finalRollerRearAxisX.cathode.inPos) OR ("Unit1.Em6.ControlNodes".cm.softCam.finalRollerFrontAxisX.anode.inPos AND "Unit1.Em6.ControlNodes".cm.softCam.finalRollerRearAxisX.anode.inPos),
                           int2 := "Unit1.Em6.ControlNodes".emRelations.em4.softCam.anodeMainPnP2AxisX.alignTablePos.inPos OR "Unit1.Em6.ControlNodes".emRelations.em4.softCam.anodeMainPnP2AxisX.stackTablePos.inPos OR "Unit1.Em6.ControlNodes".emRelations.em4.softCam.anodeMainPnP2AxisZ.upPos.inPos,
                           int3 := "Unit1.Em6.ControlNodes".emRelations.em5.softCam.cathodeMainPnP2AxisX.alignTablePos.inPos OR "Unit1.Em6.ControlNodes".emRelations.em5.softCam.cathodeMainPnP2AxisX.stackTablePos.inPos OR "Unit1.Em6.ControlNodes".emRelations.em5.softCam.cathodeMainPnP2AxisZ.upPos.inPos,
                           commands := "Unit1.Em6.HmiInterface".cmMendrelAnodeRearAxisY.commands,
                           interlockOk := "Unit1.Em6.ControlNodes".cm.Interlock.mendrelAnodeRearAxisY.source.posAbsolute,
                           intOut := "Unit1.Em6.HmiInterface".intCondition.Axis_25.Jog.intOut);
   #_w1 := NOT (NOT "Unit1.Em6.ControlNodes".stackTable."step".action1[151] AND NOT "Unit1.Em6.ControlNodes".stackTable."step".action1[2221] AND NOT "Unit1.Em6.ControlNodes".stackTable."step".action1[440]) AND "Unit1.Em6.ControlNodes".cm.Interlock.mendrelAnodeRearAxisY.source.posAbsolute[1];
   IF #_w1 THEN "Unit1.Em6.ControlNodes".cmMendrelAnodeRearAxisY.commands.selectSetPosition := 1; END_IF;
   "Unit1.Em6.ControlNodes".cm.Command.mendrelAnodeRearAxisY.posAbsolute[1] := #_w1;
END_REGION

REGION Network 149: CmMendrelAnodeRearAxisY Position Absolute Position2
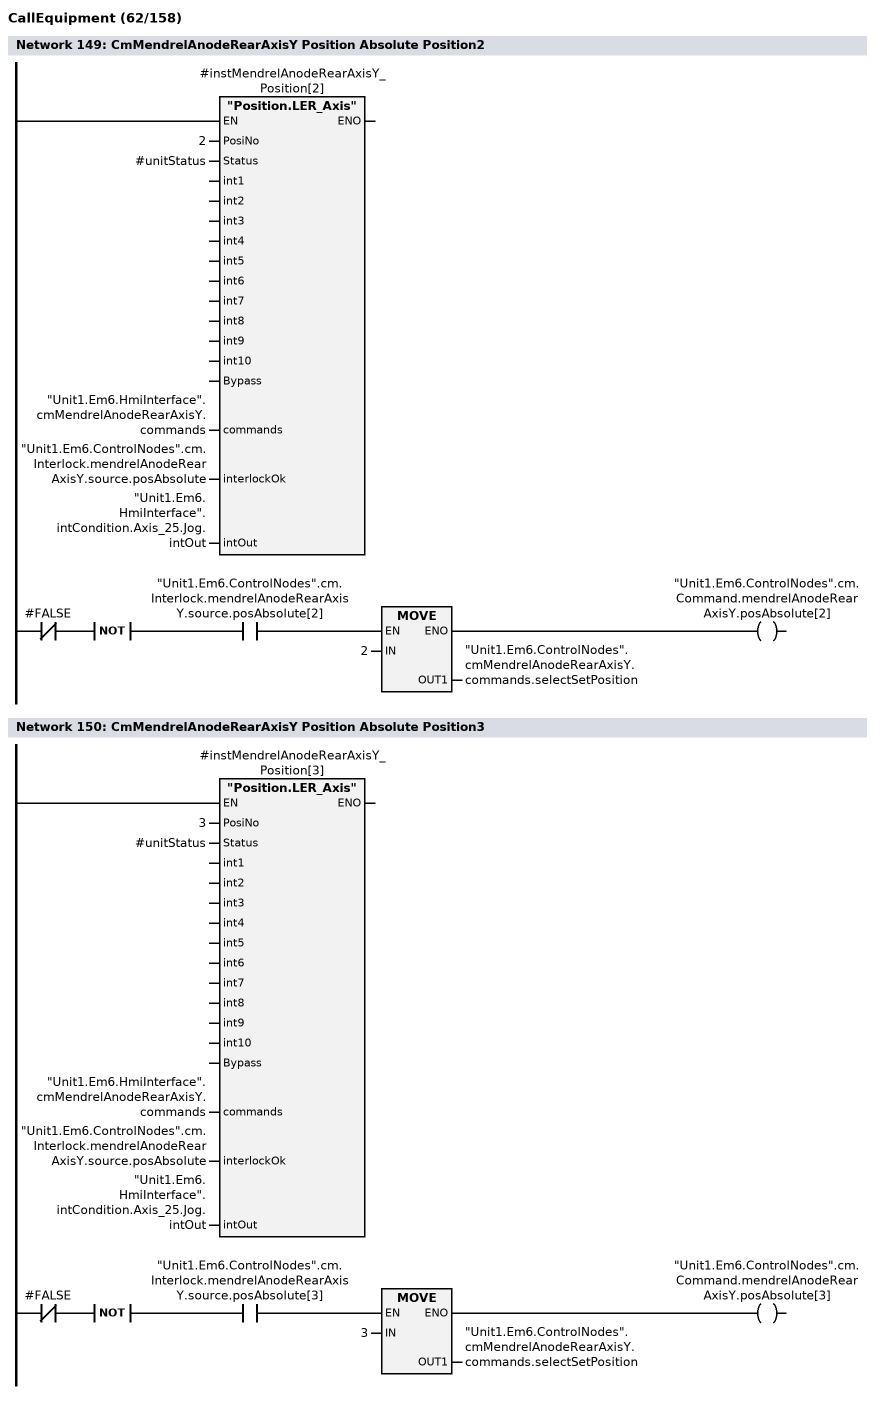
   RUNG wire#powerrail
      #instMendrelAnodeRearAxisY_Position[2](PosiNo := 2, Status := #unitStatus, int1 :=, int2 :=, int3 :=, int4 :=, int5 :=, int6 :=, int7 :=, int8 :=, int9 :=, int10 :=, Bypass :=, commands := "Unit1.Em6.HmiInterface".cmMendrelAnodeRearAxisY.commands, interlockOk := "Unit1.Em6.ControlNodes".cm.Interlock.mendrelAnodeRearAxisY.source.posAbsolute, intOut := "Unit1.Em6.HmiInterface".intCondition.Axis_25.Jog.intOut)
   END_RUNG
   RUNG wire#powerrail
      I_Contact( #FALSE )
      Not()
      Contact( "Unit1.Em6.ControlNodes".cm.Interlock.mendrelAnodeRearAxisY.source.posAbsolute[2] )
      Move(in := 2, out1 => "Unit1.Em6.ControlNodes".cmMendrelAnodeRearAxisY.commands.selectSetPosition)
      Coil( "Unit1.Em6.ControlNodes".cm.Command.mendrelAnodeRearAxisY.posAbsolute[2] )
   END_RUNG
   // the same network as SCL:
   #instMendrelAnodeRearAxisY_Position[2](PosiNo := 2,   // "Position.LER_Axis"
                           Status := #unitStatus,
                           commands := "Unit1.Em6.HmiInterface".cmMendrelAnodeRearAxisY.commands,
                           interlockOk := "Unit1.Em6.ControlNodes".cm.Interlock.mendrelAnodeRearAxisY.source.posAbsolute,
                           intOut := "Unit1.Em6.HmiInterface".intCondition.Axis_25.Jog.intOut);
   #_w1 := NOT (NOT #FALSE) AND "Unit1.Em6.ControlNodes".cm.Interlock.mendrelAnodeRearAxisY.source.posAbsolute[2];
   IF #_w1 THEN "Unit1.Em6.ControlNodes".cmMendrelAnodeRearAxisY.commands.selectSetPosition := 2; END_IF;
   "Unit1.Em6.ControlNodes".cm.Command.mendrelAnodeRearAxisY.posAbsolute[2] := #_w1;
END_REGION

REGION Network 150: CmMendrelAnodeRearAxisY Position Absolute Position3
   RUNG wire#powerrail
      #instMendrelAnodeRearAxisY_Position[3](PosiNo := 3, Status := #unitStatus, int1 :=, int2 :=, int3 :=, int4 :=, int5 :=, int6 :=, int7 :=, int8 :=, int9 :=, int10 :=, Bypass :=, commands := "Unit1.Em6.HmiInterface".cmMendrelAnodeRearAxisY.commands, interlockOk := "Unit1.Em6.ControlNodes".cm.Interlock.mendrelAnodeRearAxisY.source.posAbsolute, intOut := "Unit1.Em6.HmiInterface".intCondition.Axis_25.Jog.intOut)
   END_RUNG
   RUNG wire#powerrail
      I_Contact( #FALSE )
      Not()
      Contact( "Unit1.Em6.ControlNodes".cm.Interlock.mendrelAnodeRearAxisY.source.posAbsolute[3] )
      Move(in := 3, out1 => "Unit1.Em6.ControlNodes".cmMendrelAnodeRearAxisY.commands.selectSetPosition)
      Coil( "Unit1.Em6.ControlNodes".cm.Command.mendrelAnodeRearAxisY.posAbsolute[3] )
   END_RUNG
   // the same network as SCL:
   #instMendrelAnodeRearAxisY_Position[3](PosiNo := 3,   // "Position.LER_Axis"
                           Status := #unitStatus,
                           commands := "Unit1.Em6.HmiInterface".cmMendrelAnodeRearAxisY.commands,
                           interlockOk := "Unit1.Em6.ControlNodes".cm.Interlock.mendrelAnodeRearAxisY.source.posAbsolute,
                           intOut := "Unit1.Em6.HmiInterface".intCondition.Axis_25.Jog.intOut);
   #_w1 := NOT (NOT #FALSE) AND "Unit1.Em6.ControlNodes".cm.Interlock.mendrelAnodeRearAxisY.source.posAbsolute[3];
   IF #_w1 THEN "Unit1.Em6.ControlNodes".cmMendrelAnodeRearAxisY.commands.selectSetPosition := 3; END_IF;
   "Unit1.Em6.ControlNodes".cm.Command.mendrelAnodeRearAxisY.posAbsolute[3] := #_w1;
END_REGION

REGION Network 151: CmMendrelAnodeRearAxisY Position Absolute Position4
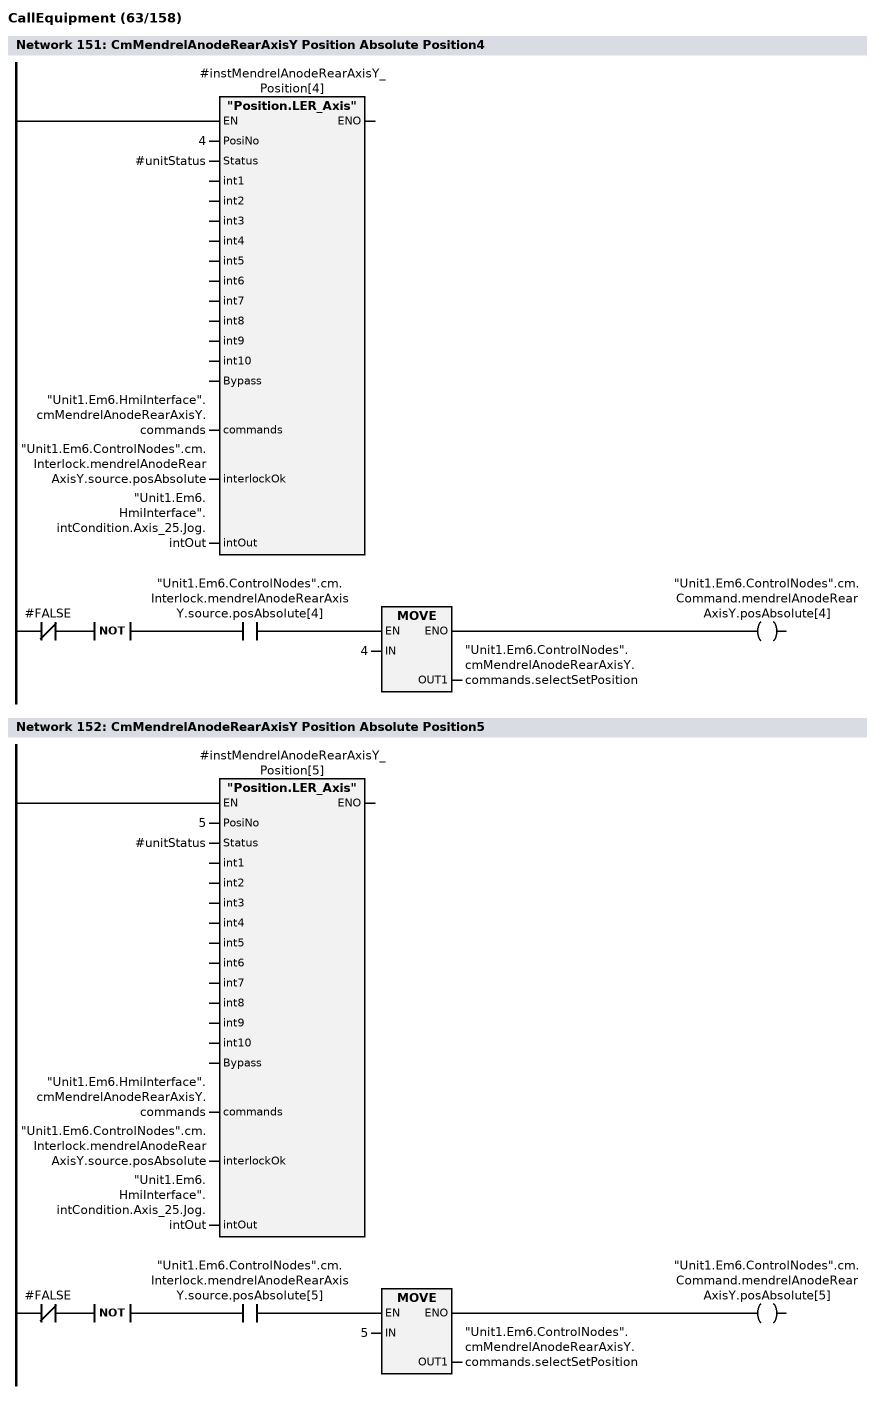
   RUNG wire#powerrail
      #instMendrelAnodeRearAxisY_Position[4](PosiNo := 4, Status := #unitStatus, int1 :=, int2 :=, int3 :=, int4 :=, int5 :=, int6 :=, int7 :=, int8 :=, int9 :=, int10 :=, Bypass :=, commands := "Unit1.Em6.HmiInterface".cmMendrelAnodeRearAxisY.commands, interlockOk := "Unit1.Em6.ControlNodes".cm.Interlock.mendrelAnodeRearAxisY.source.posAbsolute, intOut := "Unit1.Em6.HmiInterface".intCondition.Axis_25.Jog.intOut)
   END_RUNG
   RUNG wire#powerrail
      I_Contact( #FALSE )
      Not()
      Contact( "Unit1.Em6.ControlNodes".cm.Interlock.mendrelAnodeRearAxisY.source.posAbsolute[4] )
      Move(in := 4, out1 => "Unit1.Em6.ControlNodes".cmMendrelAnodeRearAxisY.commands.selectSetPosition)
      Coil( "Unit1.Em6.ControlNodes".cm.Command.mendrelAnodeRearAxisY.posAbsolute[4] )
   END_RUNG
   // the same network as SCL:
   #instMendrelAnodeRearAxisY_Position[4](PosiNo := 4,   // "Position.LER_Axis"
                           Status := #unitStatus,
                           commands := "Unit1.Em6.HmiInterface".cmMendrelAnodeRearAxisY.commands,
                           interlockOk := "Unit1.Em6.ControlNodes".cm.Interlock.mendrelAnodeRearAxisY.source.posAbsolute,
                           intOut := "Unit1.Em6.HmiInterface".intCondition.Axis_25.Jog.intOut);
   #_w1 := NOT (NOT #FALSE) AND "Unit1.Em6.ControlNodes".cm.Interlock.mendrelAnodeRearAxisY.source.posAbsolute[4];
   IF #_w1 THEN "Unit1.Em6.ControlNodes".cmMendrelAnodeRearAxisY.commands.selectSetPosition := 4; END_IF;
   "Unit1.Em6.ControlNodes".cm.Command.mendrelAnodeRearAxisY.posAbsolute[4] := #_w1;
END_REGION

REGION Network 152: CmMendrelAnodeRearAxisY Position Absolute Position5
   RUNG wire#powerrail
      #instMendrelAnodeRearAxisY_Position[5](PosiNo := 5, Status := #unitStatus, int1 :=, int2 :=, int3 :=, int4 :=, int5 :=, int6 :=, int7 :=, int8 :=, int9 :=, int10 :=, Bypass :=, commands := "Unit1.Em6.HmiInterface".cmMendrelAnodeRearAxisY.commands, interlockOk := "Unit1.Em6.ControlNodes".cm.Interlock.mendrelAnodeRearAxisY.source.posAbsolute, intOut := "Unit1.Em6.HmiInterface".intCondition.Axis_25.Jog.intOut)
   END_RUNG
   RUNG wire#powerrail
      I_Contact( #FALSE )
      Not()
      Contact( "Unit1.Em6.ControlNodes".cm.Interlock.mendrelAnodeRearAxisY.source.posAbsolute[5] )
      Move(in := 5, out1 => "Unit1.Em6.ControlNodes".cmMendrelAnodeRearAxisY.commands.selectSetPosition)
      Coil( "Unit1.Em6.ControlNodes".cm.Command.mendrelAnodeRearAxisY.posAbsolute[5] )
   END_RUNG
   // the same network as SCL:
   #instMendrelAnodeRearAxisY_Position[5](PosiNo := 5,   // "Position.LER_Axis"
                           Status := #unitStatus,
                           commands := "Unit1.Em6.HmiInterface".cmMendrelAnodeRearAxisY.commands,
                           interlockOk := "Unit1.Em6.ControlNodes".cm.Interlock.mendrelAnodeRearAxisY.source.posAbsolute,
                           intOut := "Unit1.Em6.HmiInterface".intCondition.Axis_25.Jog.intOut);
   #_w1 := NOT (NOT #FALSE) AND "Unit1.Em6.ControlNodes".cm.Interlock.mendrelAnodeRearAxisY.source.posAbsolute[5];
   IF #_w1 THEN "Unit1.Em6.ControlNodes".cmMendrelAnodeRearAxisY.commands.selectSetPosition := 5; END_IF;
   "Unit1.Em6.ControlNodes".cm.Command.mendrelAnodeRearAxisY.posAbsolute[5] := #_w1;
END_REGION

REGION Network 153: CmMendrelAnodeRearAxisY Summary Command
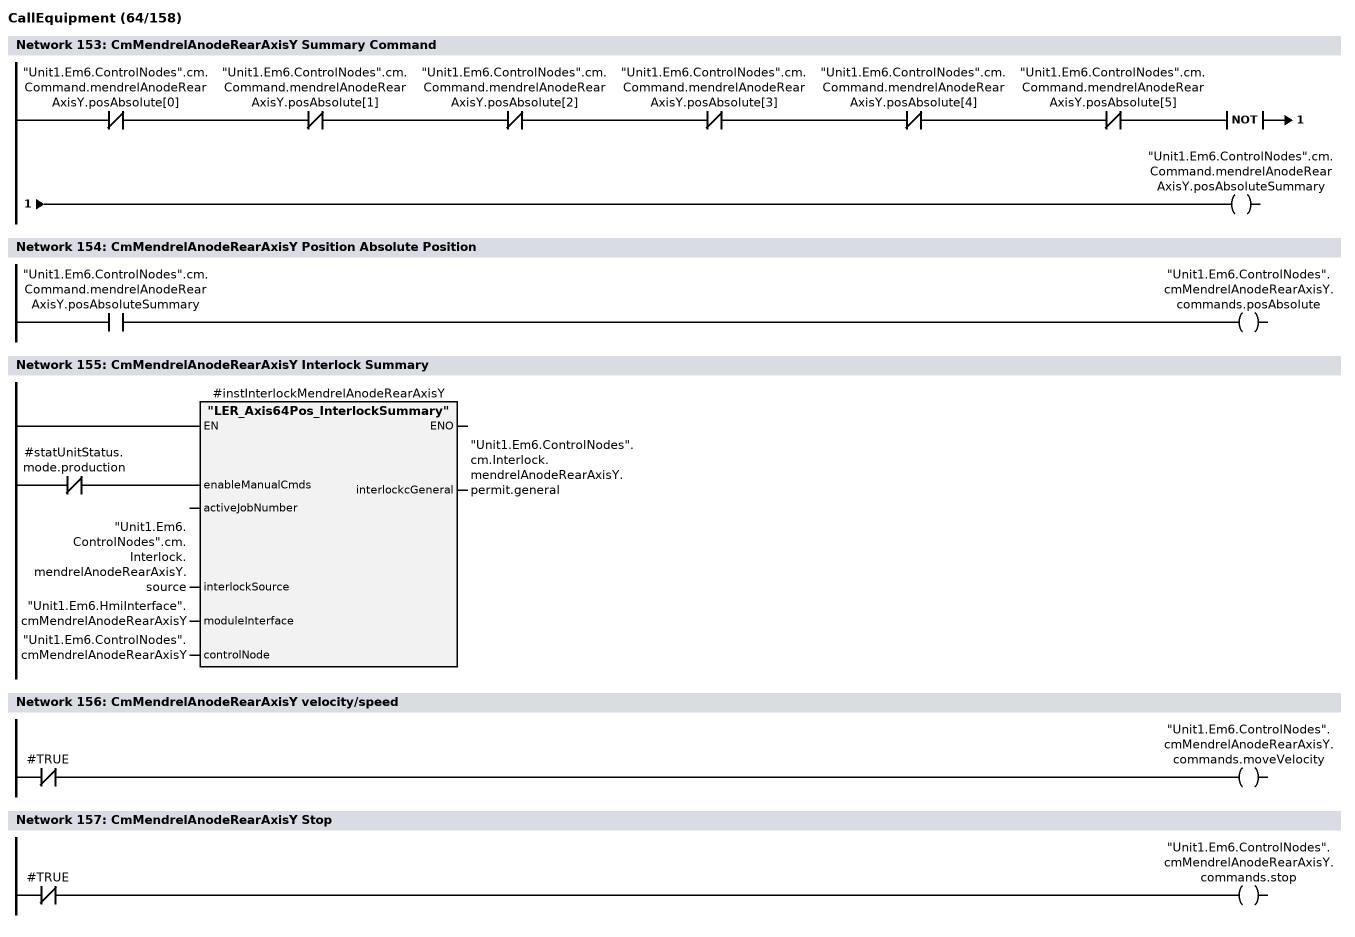
   RUNG wire#powerrail
      I_Contact( "Unit1.Em6.ControlNodes".cm.Command.mendrelAnodeRearAxisY.posAbsolute[0] )
      I_Contact( "Unit1.Em6.ControlNodes".cm.Command.mendrelAnodeRearAxisY.posAbsolute[1] )
      I_Contact( "Unit1.Em6.ControlNodes".cm.Command.mendrelAnodeRearAxisY.posAbsolute[2] )
      I_Contact( "Unit1.Em6.ControlNodes".cm.Command.mendrelAnodeRearAxisY.posAbsolute[3] )
      I_Contact( "Unit1.Em6.ControlNodes".cm.Command.mendrelAnodeRearAxisY.posAbsolute[4] )
      I_Contact( "Unit1.Em6.ControlNodes".cm.Command.mendrelAnodeRearAxisY.posAbsolute[5] )
      Not()
      Coil( "Unit1.Em6.ControlNodes".cm.Command.mendrelAnodeRearAxisY.posAbsoluteSummary )
   END_RUNG
   // the same network as SCL:
   "Unit1.Em6.ControlNodes".cm.Command.mendrelAnodeRearAxisY.posAbsoluteSummary := NOT (NOT "Unit1.Em6.ControlNodes".cm.Command.mendrelAnodeRearAxisY.posAbsolute[0] AND NOT "Unit1.Em6.ControlNodes".cm.Command.mendrelAnodeRearAxisY.posAbsolute[1] AND NOT "Unit1.Em6.ControlNodes".cm.Command.mendrelAnodeRearAxisY.posAbsolute[2] AND NOT "Unit1.Em6.ControlNodes".cm.Command.mendrelAnodeRearAxisY.posAbsolute[3] AND NOT "Unit1.Em6.ControlNodes".cm.Command.mendrelAnodeRearAxisY.posAbsolute[4] AND NOT "Unit1.Em6.ControlNodes".cm.Command.mendrelAnodeRearAxisY.posAbsolute[5]);
END_REGION

REGION Network 154: CmMendrelAnodeRearAxisY Position Absolute Position
   RUNG wire#powerrail
      Contact( "Unit1.Em6.ControlNodes".cm.Command.mendrelAnodeRearAxisY.posAbsoluteSummary )
      Coil( "Unit1.Em6.ControlNodes".cmMendrelAnodeRearAxisY.commands.posAbsolute )
   END_RUNG
   // the same network as SCL:
   "Unit1.Em6.ControlNodes".cmMendrelAnodeRearAxisY.commands.posAbsolute := "Unit1.Em6.ControlNodes".cm.Command.mendrelAnodeRearAxisY.posAbsoluteSummary;
END_REGION

REGION Network 155: CmMendrelAnodeRearAxisY Interlock Summary
   RUNG wire#powerrail
      #instInterlockMendrelAnodeRearAxisY(enableManualCmds := wire#w1, activeJobNumber :=, interlockSource := "Unit1.Em6.ControlNodes".cm.Interlock.mendrelAnodeRearAxisY.source, moduleInterface := "Unit1.Em6.HmiInterface".cmMendrelAnodeRearAxisY, controlNode := "Unit1.Em6.ControlNodes".cmMendrelAnodeRearAxisY, interlockcGeneral => "Unit1.Em6.ControlNodes".cm.Interlock.mendrelAnodeRearAxisY.permit.general)
   END_RUNG
   RUNG wire#powerrail
      I_Contact( #statUnitStatus.mode.production )
   END_RUNG wire#w1
   // the same network as SCL:
   #instInterlockMendrelAnodeRearAxisY(enableManualCmds := NOT #statUnitStatus.mode.production,   // "LER_Axis64Pos_InterlockSummary"
                           interlockSource := "Unit1.Em6.ControlNodes".cm.Interlock.mendrelAnodeRearAxisY.source,
                           moduleInterface := "Unit1.Em6.HmiInterface".cmMendrelAnodeRearAxisY,
                           controlNode := "Unit1.Em6.ControlNodes".cmMendrelAnodeRearAxisY,
                           interlockcGeneral => "Unit1.Em6.ControlNodes".cm.Interlock.mendrelAnodeRearAxisY.permit.general);
END_REGION

REGION Network 156: CmMendrelAnodeRearAxisY velocity/speed
   RUNG wire#powerrail
      I_Contact( #TRUE )
      Coil( "Unit1.Em6.ControlNodes".cmMendrelAnodeRearAxisY.commands.moveVelocity )
   END_RUNG
   // the same network as SCL:
   "Unit1.Em6.ControlNodes".cmMendrelAnodeRearAxisY.commands.moveVelocity := NOT #TRUE;
END_REGION

REGION Network 157: CmMendrelAnodeRearAxisY Stop
   RUNG wire#powerrail
      I_Contact( #TRUE )
      Coil( "Unit1.Em6.ControlNodes".cmMendrelAnodeRearAxisY.commands.stop )
   END_RUNG
   // the same network as SCL:
   "Unit1.Em6.ControlNodes".cmMendrelAnodeRearAxisY.commands.stop := NOT #TRUE;
END_REGION

REGION Network 158: Call CM Anode Mandrel Rear Y-Axis (LBC_Axis64Pos)
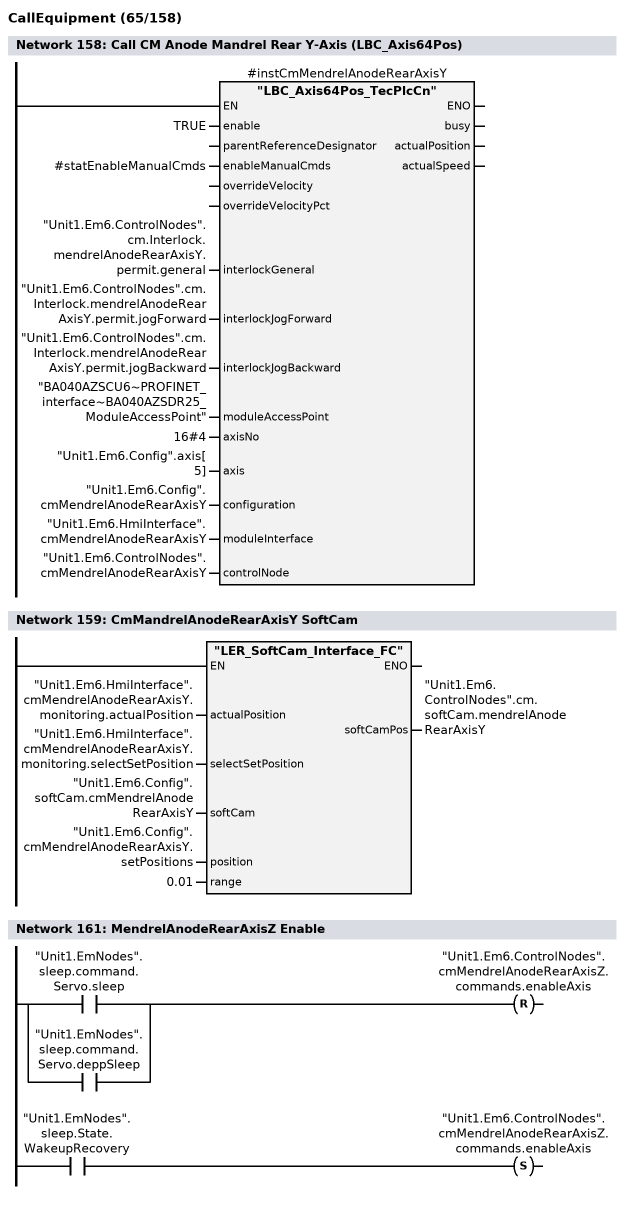
   RUNG wire#powerrail
      #instCmMendrelAnodeRearAxisY(enable := TRUE, parentReferenceDesignator :=, enableManualCmds := #statEnableManualCmds, overrideVelocity :=, overrideVelocityPct :=, interlockGeneral := "Unit1.Em6.ControlNodes".cm.Interlock.mendrelAnodeRearAxisY.permit.general, interlockJogForward := "Unit1.Em6.ControlNodes".cm.Interlock.mendrelAnodeRearAxisY.permit.jogForward, interlockJogBackward := "Unit1.Em6.ControlNodes".cm.Interlock.mendrelAnodeRearAxisY.permit.jogBackward, moduleAccessPoint := "BA040AZSCU6~PROFINET_interface~BA040AZSDR25_ModuleAccessPoint", axisNo := 16#4, axis := "Unit1.Em6.Config".axis[5], configuration := "Unit1.Em6.Config".cmMendrelAnodeRearAxisY, moduleInterface := "Unit1.Em6.HmiInterface".cmMendrelAnodeRearAxisY, controlNode := "Unit1.Em6.ControlNodes".cmMendrelAnodeRearAxisY, busy =>, actualPosition =>, actualSpeed =>)
   END_RUNG
   // the same network as SCL:
   #instCmMendrelAnodeRearAxisY(enable := TRUE,   // "LBC_Axis64Pos_TecPlcCn"
                           enableManualCmds := #statEnableManualCmds,
                           interlockGeneral := "Unit1.Em6.ControlNodes".cm.Interlock.mendrelAnodeRearAxisY.permit.general,
                           interlockJogForward := "Unit1.Em6.ControlNodes".cm.Interlock.mendrelAnodeRearAxisY.permit.jogForward,
                           interlockJogBackward := "Unit1.Em6.ControlNodes".cm.Interlock.mendrelAnodeRearAxisY.permit.jogBackward,
                           moduleAccessPoint := "BA040AZSCU6~PROFINET_interface~BA040AZSDR25_ModuleAccessPoint",
                           axisNo := 16#4,
                           axis := "Unit1.Em6.Config".axis[5],
                           configuration := "Unit1.Em6.Config".cmMendrelAnodeRearAxisY,
                           moduleInterface := "Unit1.Em6.HmiInterface".cmMendrelAnodeRearAxisY,
                           controlNode := "Unit1.Em6.ControlNodes".cmMendrelAnodeRearAxisY);
END_REGION

REGION Network 159: CmMandrelAnodeRearAxisY SoftCam
   RUNG wire#powerrail
      "LER_SoftCam_Interface_FC"(actualPosition := "Unit1.Em6.HmiInterface".cmMendrelAnodeRearAxisY.monitoring.actualPosition, selectSetPosition := "Unit1.Em6.HmiInterface".cmMendrelAnodeRearAxisY.monitoring.selectSetPosition, softCam := "Unit1.Em6.Config".softCam.cmMendrelAnodeRearAxisY, position := "Unit1.Em6.Config".cmMendrelAnodeRearAxisY.setPositions, range := 0.01, softCamPos => "Unit1.Em6.ControlNodes".cm.softCam.mendrelAnodeRearAxisY)
   END_RUNG
   // the same network as SCL:
   "LER_SoftCam_Interface_FC"(actualPosition := "Unit1.Em6.HmiInterface".cmMendrelAnodeRearAxisY.monitoring.actualPosition,
                           selectSetPosition := "Unit1.Em6.HmiInterface".cmMendrelAnodeRearAxisY.monitoring.selectSetPosition,
                           softCam := "Unit1.Em6.Config".softCam.cmMendrelAnodeRearAxisY,
                           position := "Unit1.Em6.Config".cmMendrelAnodeRearAxisY.setPositions,
                           range := 0.01,
                           softCamPos => "Unit1.Em6.ControlNodes".cm.softCam.mendrelAnodeRearAxisY);
END_REGION

REGION Network 161: MendrelAnodeRearAxisZ Enable
   RUNG wire#powerrail
      Contact( "Unit1.EmNodes".sleep.command.Servo.sleep )
      wire#w1
      R_Coil( "Unit1.Em6.ControlNodes".cmMendrelAnodeRearAxisZ.commands.enableAxis )
   END_RUNG
   RUNG wire#powerrail
      Contact( "Unit1.EmNodes".sleep.command.Servo.deppSleep )
   END_RUNG wire#w1
   RUNG wire#powerrail
      Contact( "Unit1.EmNodes".sleep.State.WakeupRecovery )
      S_Coil( "Unit1.Em6.ControlNodes".cmMendrelAnodeRearAxisZ.commands.enableAxis )
   END_RUNG
   // the same network as SCL:
   IF "Unit1.EmNodes".sleep.command.Servo.sleep OR "Unit1.EmNodes".sleep.command.Servo.deppSleep THEN
       "Unit1.Em6.ControlNodes".cmMendrelAnodeRearAxisZ.commands.enableAxis := FALSE;
   END_IF;
   IF "Unit1.EmNodes".sleep.State.WakeupRecovery THEN
       "Unit1.Em6.ControlNodes".cmMendrelAnodeRearAxisZ.commands.enableAxis := TRUE;
   END_IF;
END_REGION

REGION Network 162: CmMandrelAnodeRearAxisZ Home
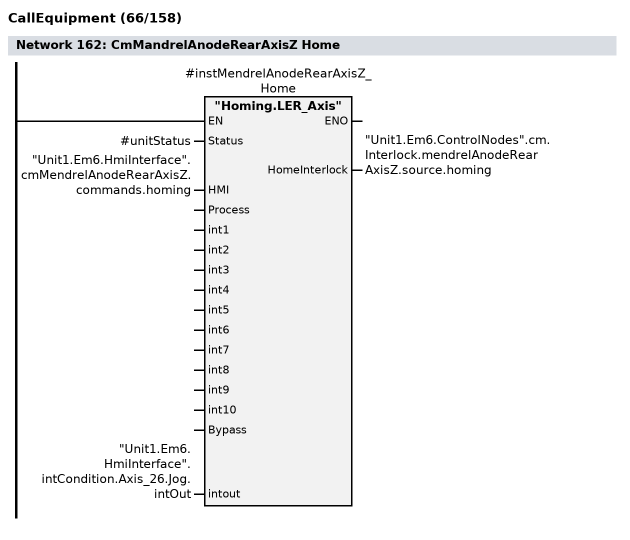
   RUNG wire#powerrail
      #instMendrelAnodeRearAxisZ_Home(Status := #unitStatus, HMI := "Unit1.Em6.HmiInterface".cmMendrelAnodeRearAxisZ.commands.homing, Process :=, int1 :=, int2 :=, int3 :=, int4 :=, int5 :=, int6 :=, int7 :=, int8 :=, int9 :=, int10 :=, Bypass :=, intout := "Unit1.Em6.HmiInterface".intCondition.Axis_26.Jog.intOut, HomeInterlock => "Unit1.Em6.ControlNodes".cm.Interlock.mendrelAnodeRearAxisZ.source.homing)
   END_RUNG
   // the same network as SCL:
   #instMendrelAnodeRearAxisZ_Home(Status := #unitStatus,   // "Homing.LER_Axis"
                           HMI := "Unit1.Em6.HmiInterface".cmMendrelAnodeRearAxisZ.commands.homing,
                           intout := "Unit1.Em6.HmiInterface".intCondition.Axis_26.Jog.intOut,
                           HomeInterlock => "Unit1.Em6.ControlNodes".cm.Interlock.mendrelAnodeRearAxisZ.source.homing);
END_REGION

REGION Network 163: CmmendrelAnodeRearAxisZ Position Absolute Jog
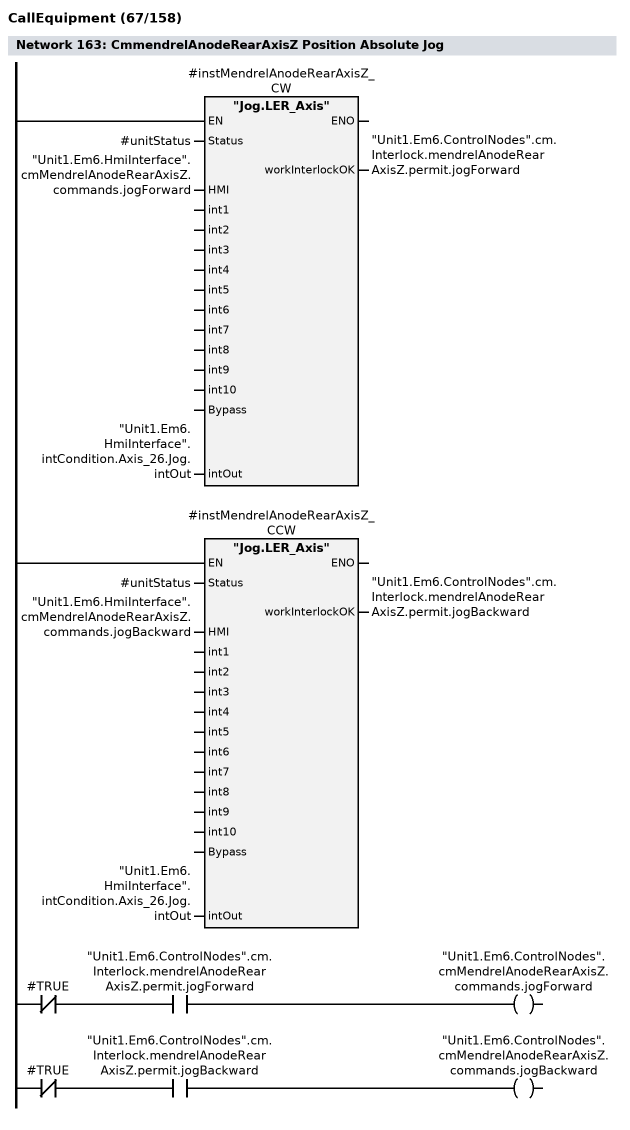
   RUNG wire#powerrail
      #instMendrelAnodeRearAxisZ_CW(Status := #unitStatus, HMI := "Unit1.Em6.HmiInterface".cmMendrelAnodeRearAxisZ.commands.jogForward, int1 :=, int2 :=, int3 :=, int4 :=, int5 :=, int6 :=, int7 :=, int8 :=, int9 :=, int10 :=, Bypass :=, intOut := "Unit1.Em6.HmiInterface".intCondition.Axis_26.Jog.intOut, workInterlockOK => "Unit1.Em6.ControlNodes".cm.Interlock.mendrelAnodeRearAxisZ.permit.jogForward)
   END_RUNG
   RUNG wire#powerrail
      #instMendrelAnodeRearAxisZ_CCW(Status := #unitStatus, HMI := "Unit1.Em6.HmiInterface".cmMendrelAnodeRearAxisZ.commands.jogBackward, int1 :=, int2 :=, int3 :=, int4 :=, int5 :=, int6 :=, int7 :=, int8 :=, int9 :=, int10 :=, Bypass :=, intOut := "Unit1.Em6.HmiInterface".intCondition.Axis_26.Jog.intOut, workInterlockOK => "Unit1.Em6.ControlNodes".cm.Interlock.mendrelAnodeRearAxisZ.permit.jogBackward)
   END_RUNG
   RUNG wire#powerrail
      I_Contact( #TRUE )
      Contact( "Unit1.Em6.ControlNodes".cm.Interlock.mendrelAnodeRearAxisZ.permit.jogForward )
      Coil( "Unit1.Em6.ControlNodes".cmMendrelAnodeRearAxisZ.commands.jogForward )
   END_RUNG
   RUNG wire#powerrail
      I_Contact( #TRUE )
      Contact( "Unit1.Em6.ControlNodes".cm.Interlock.mendrelAnodeRearAxisZ.permit.jogBackward )
      Coil( "Unit1.Em6.ControlNodes".cmMendrelAnodeRearAxisZ.commands.jogBackward )
   END_RUNG
   // the same network as SCL:
   #instMendrelAnodeRearAxisZ_CW(Status := #unitStatus,   // "Jog.LER_Axis"
                           HMI := "Unit1.Em6.HmiInterface".cmMendrelAnodeRearAxisZ.commands.jogForward,
                           intOut := "Unit1.Em6.HmiInterface".intCondition.Axis_26.Jog.intOut,
                           workInterlockOK => "Unit1.Em6.ControlNodes".cm.Interlock.mendrelAnodeRearAxisZ.permit.jogForward);
   #instMendrelAnodeRearAxisZ_CCW(Status := #unitStatus,   // "Jog.LER_Axis"
                           HMI := "Unit1.Em6.HmiInterface".cmMendrelAnodeRearAxisZ.commands.jogBackward,
                           intOut := "Unit1.Em6.HmiInterface".intCondition.Axis_26.Jog.intOut,
                           workInterlockOK => "Unit1.Em6.ControlNodes".cm.Interlock.mendrelAnodeRearAxisZ.permit.jogBackward);
   "Unit1.Em6.ControlNodes".cmMendrelAnodeRearAxisZ.commands.jogForward := NOT #TRUE AND "Unit1.Em6.ControlNodes".cm.Interlock.mendrelAnodeRearAxisZ.permit.jogForward;
   "Unit1.Em6.ControlNodes".cmMendrelAnodeRearAxisZ.commands.jogBackward := NOT #TRUE AND "Unit1.Em6.ControlNodes".cm.Interlock.mendrelAnodeRearAxisZ.permit.jogBackward;
END_REGION

REGION Network 164: CmmendrelAnodeRearAxisZ Position Absolute Position0
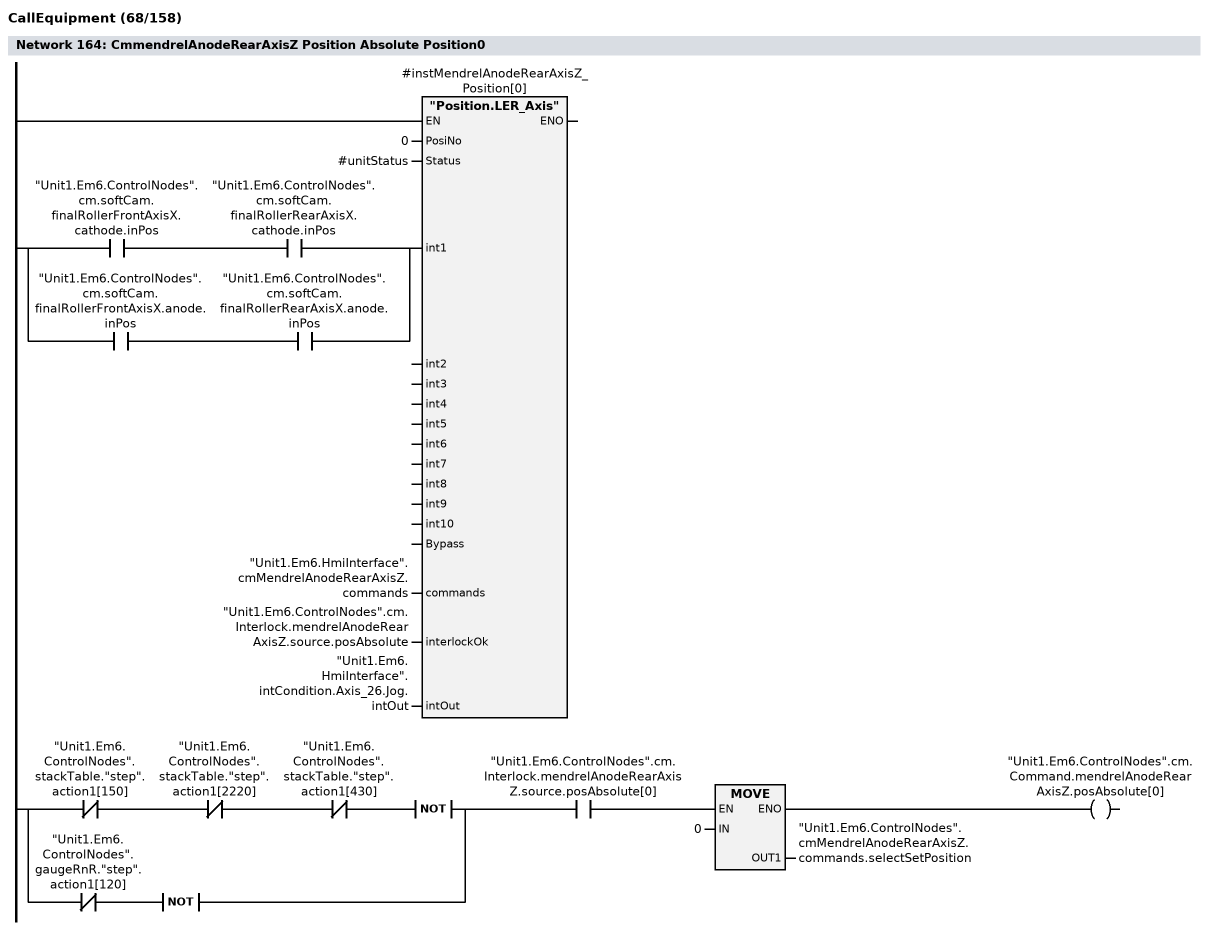
   RUNG wire#powerrail
      #instMendrelAnodeRearAxisZ_Position[0](int1 := wire#w1, PosiNo := 0, Status := #unitStatus, int2 :=, int3 :=, int4 :=, int5 :=, int6 :=, int7 :=, int8 :=, int9 :=, int10 :=, Bypass :=, commands := "Unit1.Em6.HmiInterface".cmMendrelAnodeRearAxisZ.commands, interlockOk := "Unit1.Em6.ControlNodes".cm.Interlock.mendrelAnodeRearAxisZ.source.posAbsolute, intOut := "Unit1.Em6.HmiInterface".intCondition.Axis_26.Jog.intOut)
   END_RUNG
   RUNG wire#powerrail
      Contact( "Unit1.Em6.ControlNodes".cm.softCam.finalRollerFrontAxisX.cathode.inPos )
      Contact( "Unit1.Em6.ControlNodes".cm.softCam.finalRollerRearAxisX.cathode.inPos )
   END_RUNG wire#w1
   RUNG wire#powerrail
      Contact( "Unit1.Em6.ControlNodes".cm.softCam.finalRollerFrontAxisX.anode.inPos )
      Contact( "Unit1.Em6.ControlNodes".cm.softCam.finalRollerRearAxisX.anode.inPos )
   END_RUNG wire#w1
   RUNG wire#powerrail
      I_Contact( "Unit1.Em6.ControlNodes".stackTable."step".action1[150] )
      I_Contact( "Unit1.Em6.ControlNodes".stackTable."step".action1[2220] )
      I_Contact( "Unit1.Em6.ControlNodes".stackTable."step".action1[430] )
      Not()
      wire#w2
      Contact( "Unit1.Em6.ControlNodes".cm.Interlock.mendrelAnodeRearAxisZ.source.posAbsolute[0] )
      Move(in := 0, out1 => "Unit1.Em6.ControlNodes".cmMendrelAnodeRearAxisZ.commands.selectSetPosition)
      Coil( "Unit1.Em6.ControlNodes".cm.Command.mendrelAnodeRearAxisZ.posAbsolute[0] )
   END_RUNG
   RUNG wire#powerrail
      I_Contact( "Unit1.Em6.ControlNodes".gaugeRnR."step".action1[120] )
      Not()
   END_RUNG wire#w2
   // the same network as SCL:
   #instMendrelAnodeRearAxisZ_Position[0](PosiNo := 0,   // "Position.LER_Axis"
                           Status := #unitStatus,
                           int1 := ("Unit1.Em6.ControlNodes".cm.softCam.finalRollerFrontAxisX.cathode.inPos AND "Unit1.Em6.ControlNodes".cm.softCam.finalRollerRearAxisX.cathode.inPos) OR ("Unit1.Em6.ControlNodes".cm.softCam.finalRollerFrontAxisX.anode.inPos AND "Unit1.Em6.ControlNodes".cm.softCam.finalRollerRearAxisX.anode.inPos),
                           commands := "Unit1.Em6.HmiInterface".cmMendrelAnodeRearAxisZ.commands,
                           interlockOk := "Unit1.Em6.ControlNodes".cm.Interlock.mendrelAnodeRearAxisZ.source.posAbsolute,
                           intOut := "Unit1.Em6.HmiInterface".intCondition.Axis_26.Jog.intOut);
   #_w1 := (NOT (NOT "Unit1.Em6.ControlNodes".stackTable."step".action1[150] AND NOT "Unit1.Em6.ControlNodes".stackTable."step".action1[2220] AND NOT "Unit1.Em6.ControlNodes".stackTable."step".action1[430]) OR NOT (NOT "Unit1.Em6.ControlNodes".gaugeRnR."step".action1[120])) AND "Unit1.Em6.ControlNodes".cm.Interlock.mendrelAnodeRearAxisZ.source.posAbsolute[0];
   IF #_w1 THEN "Unit1.Em6.ControlNodes".cmMendrelAnodeRearAxisZ.commands.selectSetPosition := 0; END_IF;
   "Unit1.Em6.ControlNodes".cm.Command.mendrelAnodeRearAxisZ.posAbsolute[0] := #_w1;
END_REGION

REGION Network 165: CmmendrelAnodeRearAxisZ Position Absolute Position1
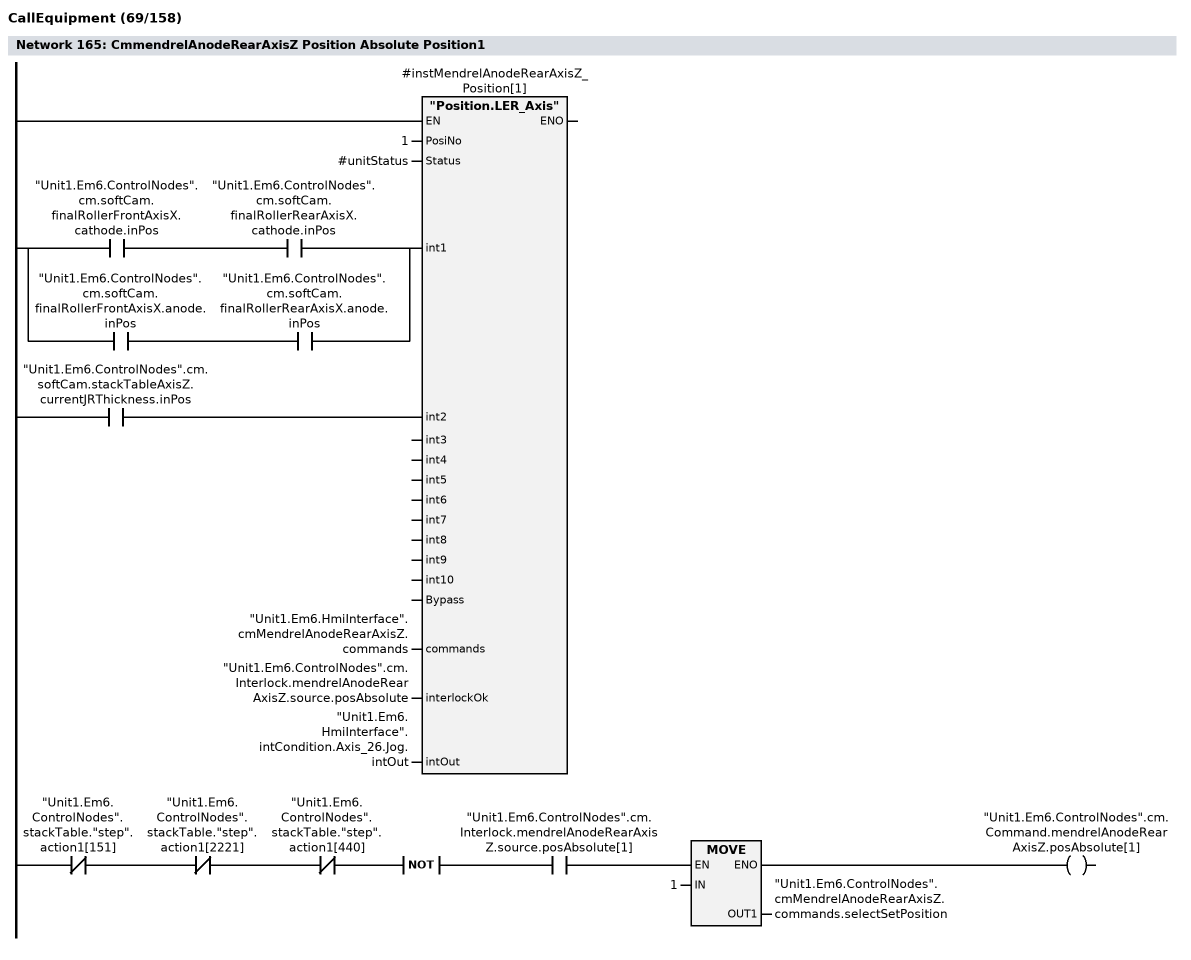
   RUNG wire#powerrail
      #instMendrelAnodeRearAxisZ_Position[1](int1 := wire#w1, int2 := wire#w2, PosiNo := 1, Status := #unitStatus, int3 :=, int4 :=, int5 :=, int6 :=, int7 :=, int8 :=, int9 :=, int10 :=, Bypass :=, commands := "Unit1.Em6.HmiInterface".cmMendrelAnodeRearAxisZ.commands, interlockOk := "Unit1.Em6.ControlNodes".cm.Interlock.mendrelAnodeRearAxisZ.source.posAbsolute, intOut := "Unit1.Em6.HmiInterface".intCondition.Axis_26.Jog.intOut)
   END_RUNG
   RUNG wire#powerrail
      Contact( "Unit1.Em6.ControlNodes".cm.softCam.finalRollerFrontAxisX.cathode.inPos )
      Contact( "Unit1.Em6.ControlNodes".cm.softCam.finalRollerRearAxisX.cathode.inPos )
   END_RUNG wire#w1
   RUNG wire#powerrail
      Contact( "Unit1.Em6.ControlNodes".cm.softCam.finalRollerFrontAxisX.anode.inPos )
      Contact( "Unit1.Em6.ControlNodes".cm.softCam.finalRollerRearAxisX.anode.inPos )
   END_RUNG wire#w1
   RUNG wire#powerrail
      Contact( "Unit1.Em6.ControlNodes".cm.softCam.stackTableAxisZ.currentJRThickness.inPos )
   END_RUNG wire#w2
   RUNG wire#powerrail
      I_Contact( "Unit1.Em6.ControlNodes".stackTable."step".action1[151] )
      I_Contact( "Unit1.Em6.ControlNodes".stackTable."step".action1[2221] )
      I_Contact( "Unit1.Em6.ControlNodes".stackTable."step".action1[440] )
      Not()
      Contact( "Unit1.Em6.ControlNodes".cm.Interlock.mendrelAnodeRearAxisZ.source.posAbsolute[1] )
      Move(in := 1, out1 => "Unit1.Em6.ControlNodes".cmMendrelAnodeRearAxisZ.commands.selectSetPosition)
      Coil( "Unit1.Em6.ControlNodes".cm.Command.mendrelAnodeRearAxisZ.posAbsolute[1] )
   END_RUNG
   // the same network as SCL:
   #instMendrelAnodeRearAxisZ_Position[1](PosiNo := 1,   // "Position.LER_Axis"
                           Status := #unitStatus,
                           int1 := ("Unit1.Em6.ControlNodes".cm.softCam.finalRollerFrontAxisX.cathode.inPos AND "Unit1.Em6.ControlNodes".cm.softCam.finalRollerRearAxisX.cathode.inPos) OR ("Unit1.Em6.ControlNodes".cm.softCam.finalRollerFrontAxisX.anode.inPos AND "Unit1.Em6.ControlNodes".cm.softCam.finalRollerRearAxisX.anode.inPos),
                           int2 := "Unit1.Em6.ControlNodes".cm.softCam.stackTableAxisZ.currentJRThickness.inPos,
                           commands := "Unit1.Em6.HmiInterface".cmMendrelAnodeRearAxisZ.commands,
                           interlockOk := "Unit1.Em6.ControlNodes".cm.Interlock.mendrelAnodeRearAxisZ.source.posAbsolute,
                           intOut := "Unit1.Em6.HmiInterface".intCondition.Axis_26.Jog.intOut);
   #_w1 := NOT (NOT "Unit1.Em6.ControlNodes".stackTable."step".action1[151] AND NOT "Unit1.Em6.ControlNodes".stackTable."step".action1[2221] AND NOT "Unit1.Em6.ControlNodes".stackTable."step".action1[440]) AND "Unit1.Em6.ControlNodes".cm.Interlock.mendrelAnodeRearAxisZ.source.posAbsolute[1];
   IF #_w1 THEN "Unit1.Em6.ControlNodes".cmMendrelAnodeRearAxisZ.commands.selectSetPosition := 1; END_IF;
   "Unit1.Em6.ControlNodes".cm.Command.mendrelAnodeRearAxisZ.posAbsolute[1] := #_w1;
END_REGION

REGION Network 166: CmmendrelAnodeRearAxisZ Position Absolute Position2
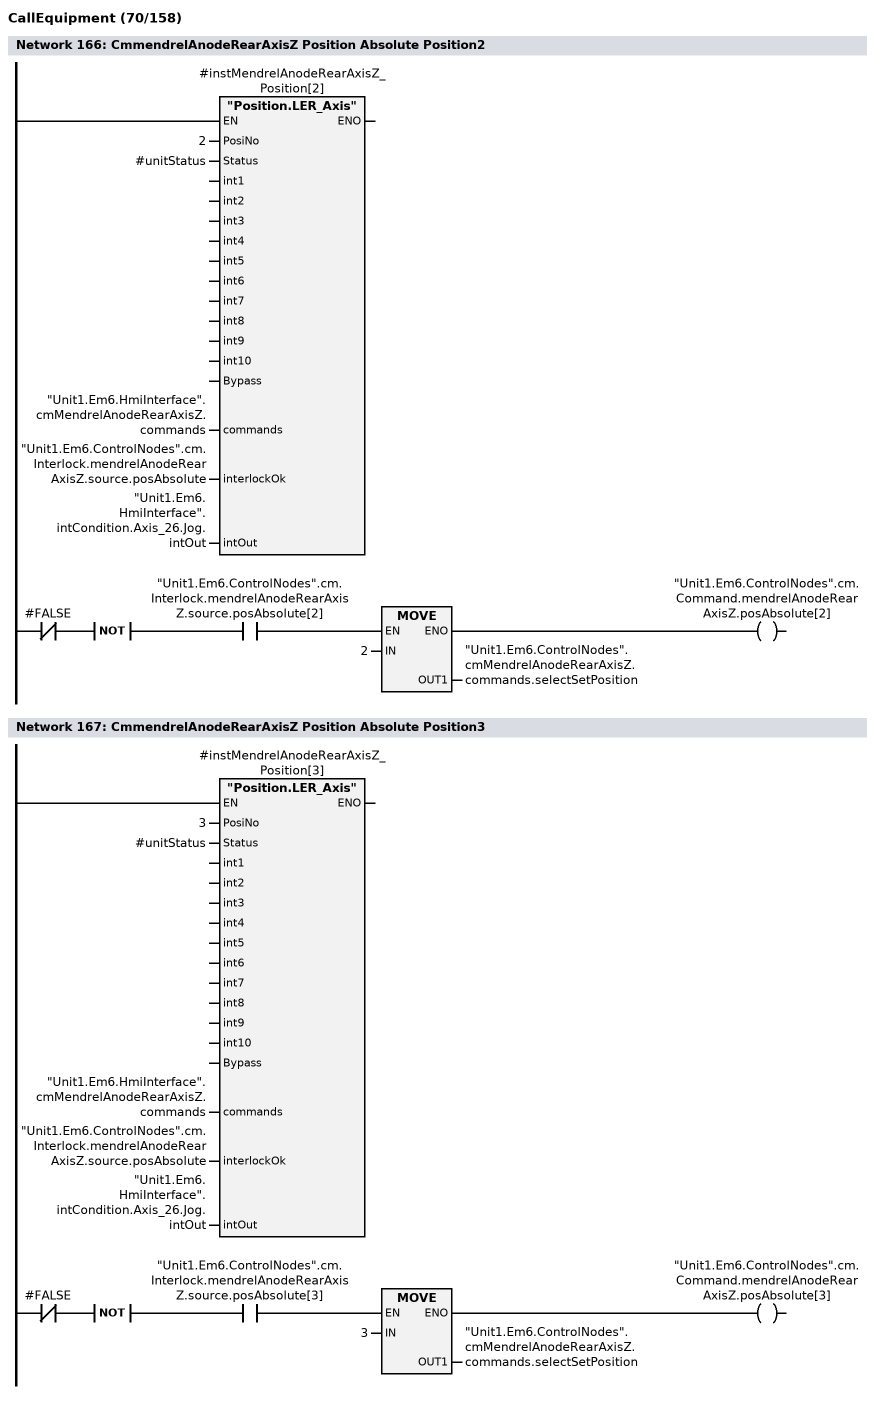
   RUNG wire#powerrail
      #instMendrelAnodeRearAxisZ_Position[2](PosiNo := 2, Status := #unitStatus, int1 :=, int2 :=, int3 :=, int4 :=, int5 :=, int6 :=, int7 :=, int8 :=, int9 :=, int10 :=, Bypass :=, commands := "Unit1.Em6.HmiInterface".cmMendrelAnodeRearAxisZ.commands, interlockOk := "Unit1.Em6.ControlNodes".cm.Interlock.mendrelAnodeRearAxisZ.source.posAbsolute, intOut := "Unit1.Em6.HmiInterface".intCondition.Axis_26.Jog.intOut)
   END_RUNG
   RUNG wire#powerrail
      I_Contact( #FALSE )
      Not()
      Contact( "Unit1.Em6.ControlNodes".cm.Interlock.mendrelAnodeRearAxisZ.source.posAbsolute[2] )
      Move(in := 2, out1 => "Unit1.Em6.ControlNodes".cmMendrelAnodeRearAxisZ.commands.selectSetPosition)
      Coil( "Unit1.Em6.ControlNodes".cm.Command.mendrelAnodeRearAxisZ.posAbsolute[2] )
   END_RUNG
   // the same network as SCL:
   #instMendrelAnodeRearAxisZ_Position[2](PosiNo := 2,   // "Position.LER_Axis"
                           Status := #unitStatus,
                           commands := "Unit1.Em6.HmiInterface".cmMendrelAnodeRearAxisZ.commands,
                           interlockOk := "Unit1.Em6.ControlNodes".cm.Interlock.mendrelAnodeRearAxisZ.source.posAbsolute,
                           intOut := "Unit1.Em6.HmiInterface".intCondition.Axis_26.Jog.intOut);
   #_w1 := NOT (NOT #FALSE) AND "Unit1.Em6.ControlNodes".cm.Interlock.mendrelAnodeRearAxisZ.source.posAbsolute[2];
   IF #_w1 THEN "Unit1.Em6.ControlNodes".cmMendrelAnodeRearAxisZ.commands.selectSetPosition := 2; END_IF;
   "Unit1.Em6.ControlNodes".cm.Command.mendrelAnodeRearAxisZ.posAbsolute[2] := #_w1;
END_REGION

REGION Network 167: CmmendrelAnodeRearAxisZ Position Absolute Position3
   RUNG wire#powerrail
      #instMendrelAnodeRearAxisZ_Position[3](PosiNo := 3, Status := #unitStatus, int1 :=, int2 :=, int3 :=, int4 :=, int5 :=, int6 :=, int7 :=, int8 :=, int9 :=, int10 :=, Bypass :=, commands := "Unit1.Em6.HmiInterface".cmMendrelAnodeRearAxisZ.commands, interlockOk := "Unit1.Em6.ControlNodes".cm.Interlock.mendrelAnodeRearAxisZ.source.posAbsolute, intOut := "Unit1.Em6.HmiInterface".intCondition.Axis_26.Jog.intOut)
   END_RUNG
   RUNG wire#powerrail
      I_Contact( #FALSE )
      Not()
      Contact( "Unit1.Em6.ControlNodes".cm.Interlock.mendrelAnodeRearAxisZ.source.posAbsolute[3] )
      Move(in := 3, out1 => "Unit1.Em6.ControlNodes".cmMendrelAnodeRearAxisZ.commands.selectSetPosition)
      Coil( "Unit1.Em6.ControlNodes".cm.Command.mendrelAnodeRearAxisZ.posAbsolute[3] )
   END_RUNG
   // the same network as SCL:
   #instMendrelAnodeRearAxisZ_Position[3](PosiNo := 3,   // "Position.LER_Axis"
                           Status := #unitStatus,
                           commands := "Unit1.Em6.HmiInterface".cmMendrelAnodeRearAxisZ.commands,
                           interlockOk := "Unit1.Em6.ControlNodes".cm.Interlock.mendrelAnodeRearAxisZ.source.posAbsolute,
                           intOut := "Unit1.Em6.HmiInterface".intCondition.Axis_26.Jog.intOut);
   #_w1 := NOT (NOT #FALSE) AND "Unit1.Em6.ControlNodes".cm.Interlock.mendrelAnodeRearAxisZ.source.posAbsolute[3];
   IF #_w1 THEN "Unit1.Em6.ControlNodes".cmMendrelAnodeRearAxisZ.commands.selectSetPosition := 3; END_IF;
   "Unit1.Em6.ControlNodes".cm.Command.mendrelAnodeRearAxisZ.posAbsolute[3] := #_w1;
END_REGION

REGION Network 168: CmmendrelAnodeRearAxisZ Position Absolute Position4
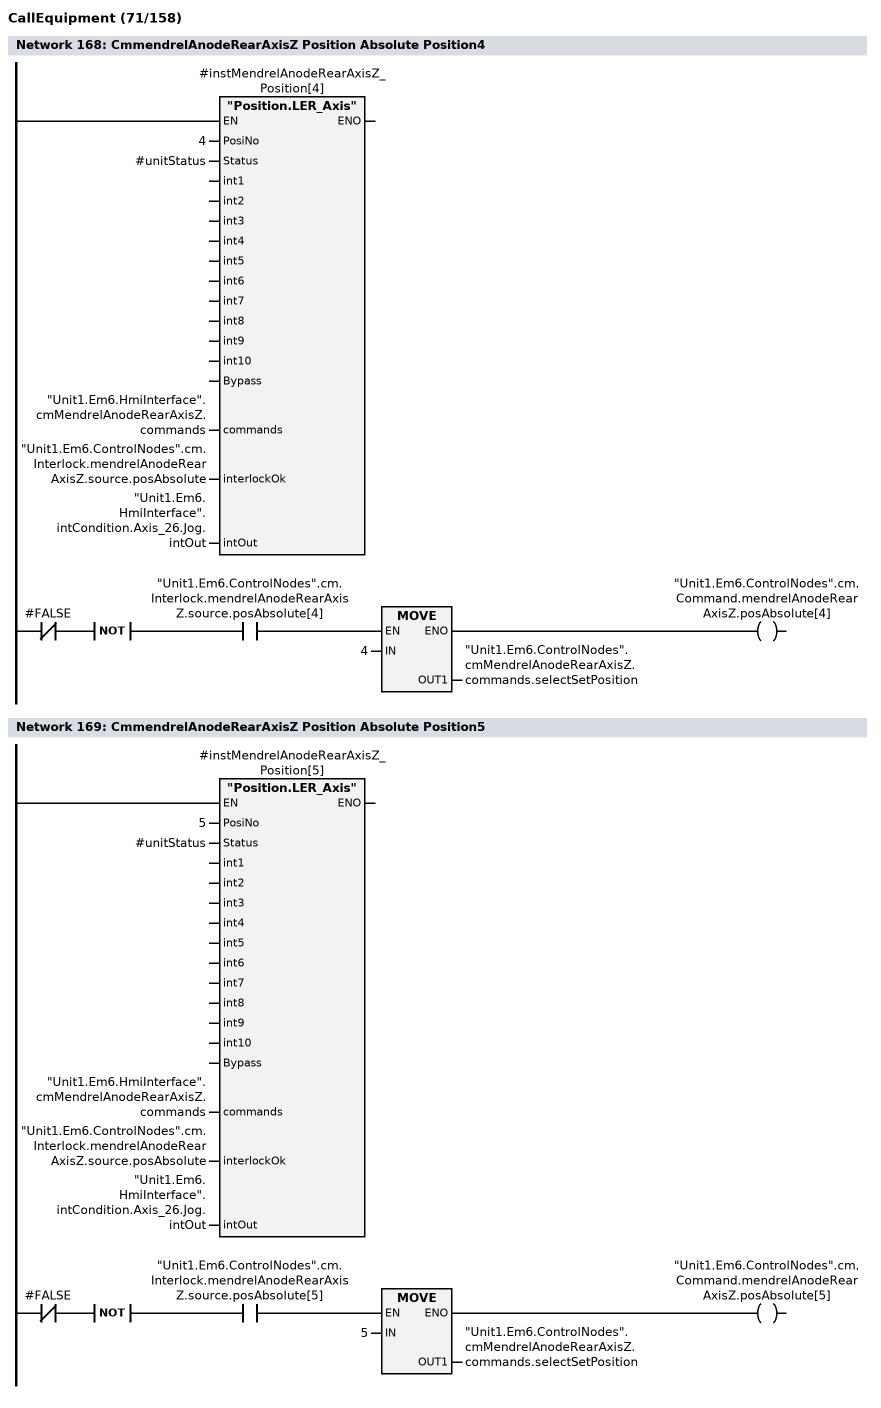
   RUNG wire#powerrail
      #instMendrelAnodeRearAxisZ_Position[4](PosiNo := 4, Status := #unitStatus, int1 :=, int2 :=, int3 :=, int4 :=, int5 :=, int6 :=, int7 :=, int8 :=, int9 :=, int10 :=, Bypass :=, commands := "Unit1.Em6.HmiInterface".cmMendrelAnodeRearAxisZ.commands, interlockOk := "Unit1.Em6.ControlNodes".cm.Interlock.mendrelAnodeRearAxisZ.source.posAbsolute, intOut := "Unit1.Em6.HmiInterface".intCondition.Axis_26.Jog.intOut)
   END_RUNG
   RUNG wire#powerrail
      I_Contact( #FALSE )
      Not()
      Contact( "Unit1.Em6.ControlNodes".cm.Interlock.mendrelAnodeRearAxisZ.source.posAbsolute[4] )
      Move(in := 4, out1 => "Unit1.Em6.ControlNodes".cmMendrelAnodeRearAxisZ.commands.selectSetPosition)
      Coil( "Unit1.Em6.ControlNodes".cm.Command.mendrelAnodeRearAxisZ.posAbsolute[4] )
   END_RUNG
   // the same network as SCL:
   #instMendrelAnodeRearAxisZ_Position[4](PosiNo := 4,   // "Position.LER_Axis"
                           Status := #unitStatus,
                           commands := "Unit1.Em6.HmiInterface".cmMendrelAnodeRearAxisZ.commands,
                           interlockOk := "Unit1.Em6.ControlNodes".cm.Interlock.mendrelAnodeRearAxisZ.source.posAbsolute,
                           intOut := "Unit1.Em6.HmiInterface".intCondition.Axis_26.Jog.intOut);
   #_w1 := NOT (NOT #FALSE) AND "Unit1.Em6.ControlNodes".cm.Interlock.mendrelAnodeRearAxisZ.source.posAbsolute[4];
   IF #_w1 THEN "Unit1.Em6.ControlNodes".cmMendrelAnodeRearAxisZ.commands.selectSetPosition := 4; END_IF;
   "Unit1.Em6.ControlNodes".cm.Command.mendrelAnodeRearAxisZ.posAbsolute[4] := #_w1;
END_REGION

REGION Network 169: CmmendrelAnodeRearAxisZ Position Absolute Position5
   RUNG wire#powerrail
      #instMendrelAnodeRearAxisZ_Position[5](PosiNo := 5, Status := #unitStatus, int1 :=, int2 :=, int3 :=, int4 :=, int5 :=, int6 :=, int7 :=, int8 :=, int9 :=, int10 :=, Bypass :=, commands := "Unit1.Em6.HmiInterface".cmMendrelAnodeRearAxisZ.commands, interlockOk := "Unit1.Em6.ControlNodes".cm.Interlock.mendrelAnodeRearAxisZ.source.posAbsolute, intOut := "Unit1.Em6.HmiInterface".intCondition.Axis_26.Jog.intOut)
   END_RUNG
   RUNG wire#powerrail
      I_Contact( #FALSE )
      Not()
      Contact( "Unit1.Em6.ControlNodes".cm.Interlock.mendrelAnodeRearAxisZ.source.posAbsolute[5] )
      Move(in := 5, out1 => "Unit1.Em6.ControlNodes".cmMendrelAnodeRearAxisZ.commands.selectSetPosition)
      Coil( "Unit1.Em6.ControlNodes".cm.Command.mendrelAnodeRearAxisZ.posAbsolute[5] )
   END_RUNG
   // the same network as SCL:
   #instMendrelAnodeRearAxisZ_Position[5](PosiNo := 5,   // "Position.LER_Axis"
                           Status := #unitStatus,
                           commands := "Unit1.Em6.HmiInterface".cmMendrelAnodeRearAxisZ.commands,
                           interlockOk := "Unit1.Em6.ControlNodes".cm.Interlock.mendrelAnodeRearAxisZ.source.posAbsolute,
                           intOut := "Unit1.Em6.HmiInterface".intCondition.Axis_26.Jog.intOut);
   #_w1 := NOT (NOT #FALSE) AND "Unit1.Em6.ControlNodes".cm.Interlock.mendrelAnodeRearAxisZ.source.posAbsolute[5];
   IF #_w1 THEN "Unit1.Em6.ControlNodes".cmMendrelAnodeRearAxisZ.commands.selectSetPosition := 5; END_IF;
   "Unit1.Em6.ControlNodes".cm.Command.mendrelAnodeRearAxisZ.posAbsolute[5] := #_w1;
END_REGION

REGION Network 170: CmmendrelAnodeRearAxisZ Summary Command
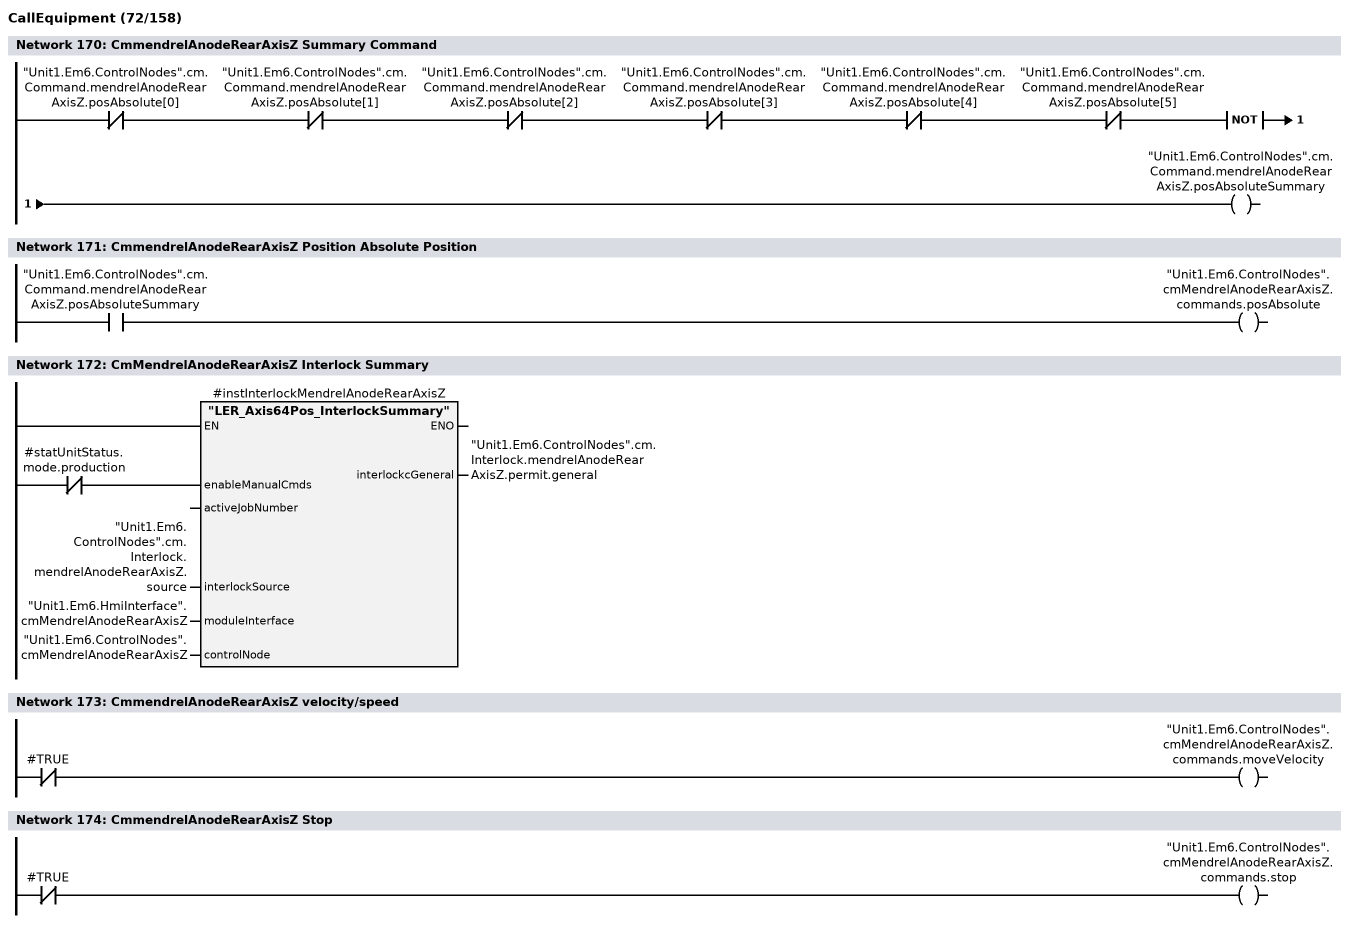
   RUNG wire#powerrail
      I_Contact( "Unit1.Em6.ControlNodes".cm.Command.mendrelAnodeRearAxisZ.posAbsolute[0] )
      I_Contact( "Unit1.Em6.ControlNodes".cm.Command.mendrelAnodeRearAxisZ.posAbsolute[1] )
      I_Contact( "Unit1.Em6.ControlNodes".cm.Command.mendrelAnodeRearAxisZ.posAbsolute[2] )
      I_Contact( "Unit1.Em6.ControlNodes".cm.Command.mendrelAnodeRearAxisZ.posAbsolute[3] )
      I_Contact( "Unit1.Em6.ControlNodes".cm.Command.mendrelAnodeRearAxisZ.posAbsolute[4] )
      I_Contact( "Unit1.Em6.ControlNodes".cm.Command.mendrelAnodeRearAxisZ.posAbsolute[5] )
      Not()
      Coil( "Unit1.Em6.ControlNodes".cm.Command.mendrelAnodeRearAxisZ.posAbsoluteSummary )
   END_RUNG
   // the same network as SCL:
   "Unit1.Em6.ControlNodes".cm.Command.mendrelAnodeRearAxisZ.posAbsoluteSummary := NOT (NOT "Unit1.Em6.ControlNodes".cm.Command.mendrelAnodeRearAxisZ.posAbsolute[0] AND NOT "Unit1.Em6.ControlNodes".cm.Command.mendrelAnodeRearAxisZ.posAbsolute[1] AND NOT "Unit1.Em6.ControlNodes".cm.Command.mendrelAnodeRearAxisZ.posAbsolute[2] AND NOT "Unit1.Em6.ControlNodes".cm.Command.mendrelAnodeRearAxisZ.posAbsolute[3] AND NOT "Unit1.Em6.ControlNodes".cm.Command.mendrelAnodeRearAxisZ.posAbsolute[4] AND NOT "Unit1.Em6.ControlNodes".cm.Command.mendrelAnodeRearAxisZ.posAbsolute[5]);
END_REGION

REGION Network 171: CmmendrelAnodeRearAxisZ Position Absolute Position
   RUNG wire#powerrail
      Contact( "Unit1.Em6.ControlNodes".cm.Command.mendrelAnodeRearAxisZ.posAbsoluteSummary )
      Coil( "Unit1.Em6.ControlNodes".cmMendrelAnodeRearAxisZ.commands.posAbsolute )
   END_RUNG
   // the same network as SCL:
   "Unit1.Em6.ControlNodes".cmMendrelAnodeRearAxisZ.commands.posAbsolute := "Unit1.Em6.ControlNodes".cm.Command.mendrelAnodeRearAxisZ.posAbsoluteSummary;
END_REGION

REGION Network 172: CmMendrelAnodeRearAxisZ Interlock Summary
   RUNG wire#powerrail
      #instInterlockMendrelAnodeRearAxisZ(enableManualCmds := wire#w1, activeJobNumber :=, interlockSource := "Unit1.Em6.ControlNodes".cm.Interlock.mendrelAnodeRearAxisZ.source, moduleInterface := "Unit1.Em6.HmiInterface".cmMendrelAnodeRearAxisZ, controlNode := "Unit1.Em6.ControlNodes".cmMendrelAnodeRearAxisZ, interlockcGeneral => "Unit1.Em6.ControlNodes".cm.Interlock.mendrelAnodeRearAxisZ.permit.general)
   END_RUNG
   RUNG wire#powerrail
      I_Contact( #statUnitStatus.mode.production )
   END_RUNG wire#w1
   // the same network as SCL:
   #instInterlockMendrelAnodeRearAxisZ(enableManualCmds := NOT #statUnitStatus.mode.production,   // "LER_Axis64Pos_InterlockSummary"
                           interlockSource := "Unit1.Em6.ControlNodes".cm.Interlock.mendrelAnodeRearAxisZ.source,
                           moduleInterface := "Unit1.Em6.HmiInterface".cmMendrelAnodeRearAxisZ,
                           controlNode := "Unit1.Em6.ControlNodes".cmMendrelAnodeRearAxisZ,
                           interlockcGeneral => "Unit1.Em6.ControlNodes".cm.Interlock.mendrelAnodeRearAxisZ.permit.general);
END_REGION

REGION Network 173: CmmendrelAnodeRearAxisZ velocity/speed
   RUNG wire#powerrail
      I_Contact( #TRUE )
      Coil( "Unit1.Em6.ControlNodes".cmMendrelAnodeRearAxisZ.commands.moveVelocity )
   END_RUNG
   // the same network as SCL:
   "Unit1.Em6.ControlNodes".cmMendrelAnodeRearAxisZ.commands.moveVelocity := NOT #TRUE;
END_REGION

REGION Network 174: CmmendrelAnodeRearAxisZ Stop
   RUNG wire#powerrail
      I_Contact( #TRUE )
      Coil( "Unit1.Em6.ControlNodes".cmMendrelAnodeRearAxisZ.commands.stop )
   END_RUNG
   // the same network as SCL:
   "Unit1.Em6.ControlNodes".cmMendrelAnodeRearAxisZ.commands.stop := NOT #TRUE;
END_REGION

REGION Network 175: Call CM Anode Mandrel Rear Z-Axis (LBC_Axis64Pos)
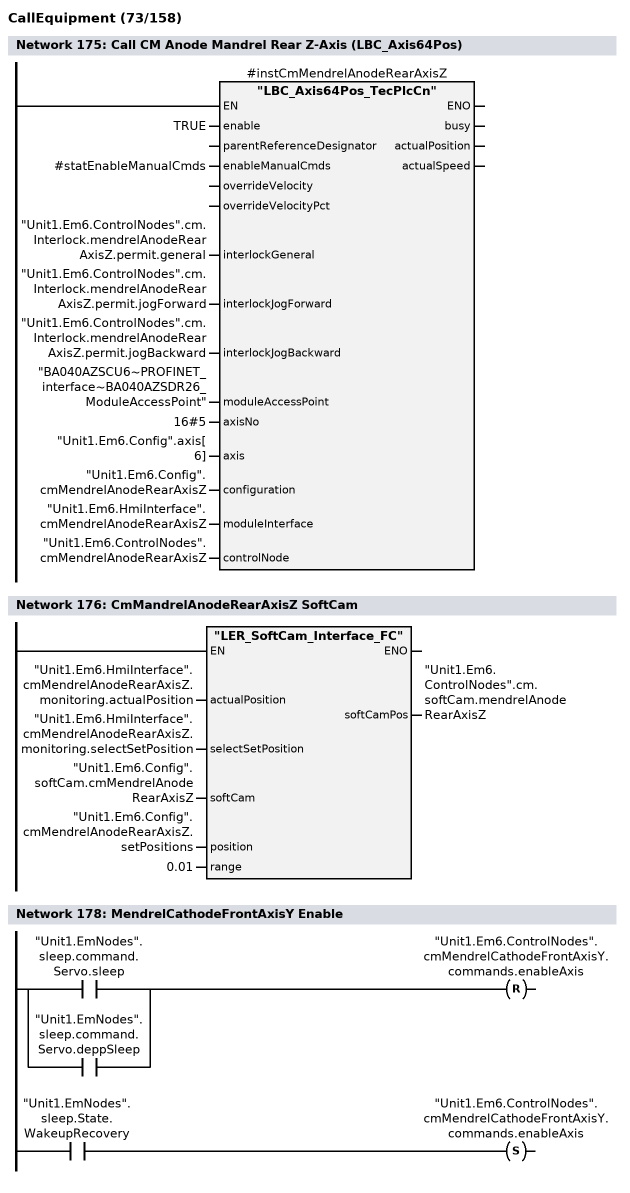
   RUNG wire#powerrail
      #instCmMendrelAnodeRearAxisZ(enable := TRUE, parentReferenceDesignator :=, enableManualCmds := #statEnableManualCmds, overrideVelocity :=, overrideVelocityPct :=, interlockGeneral := "Unit1.Em6.ControlNodes".cm.Interlock.mendrelAnodeRearAxisZ.permit.general, interlockJogForward := "Unit1.Em6.ControlNodes".cm.Interlock.mendrelAnodeRearAxisZ.permit.jogForward, interlockJogBackward := "Unit1.Em6.ControlNodes".cm.Interlock.mendrelAnodeRearAxisZ.permit.jogBackward, moduleAccessPoint := "BA040AZSCU6~PROFINET_interface~BA040AZSDR26_ModuleAccessPoint", axisNo := 16#5, axis := "Unit1.Em6.Config".axis[6], configuration := "Unit1.Em6.Config".cmMendrelAnodeRearAxisZ, moduleInterface := "Unit1.Em6.HmiInterface".cmMendrelAnodeRearAxisZ, controlNode := "Unit1.Em6.ControlNodes".cmMendrelAnodeRearAxisZ, busy =>, actualPosition =>, actualSpeed =>)
   END_RUNG
   // the same network as SCL:
   #instCmMendrelAnodeRearAxisZ(enable := TRUE,   // "LBC_Axis64Pos_TecPlcCn"
                           enableManualCmds := #statEnableManualCmds,
                           interlockGeneral := "Unit1.Em6.ControlNodes".cm.Interlock.mendrelAnodeRearAxisZ.permit.general,
                           interlockJogForward := "Unit1.Em6.ControlNodes".cm.Interlock.mendrelAnodeRearAxisZ.permit.jogForward,
                           interlockJogBackward := "Unit1.Em6.ControlNodes".cm.Interlock.mendrelAnodeRearAxisZ.permit.jogBackward,
                           moduleAccessPoint := "BA040AZSCU6~PROFINET_interface~BA040AZSDR26_ModuleAccessPoint",
                           axisNo := 16#5,
                           axis := "Unit1.Em6.Config".axis[6],
                           configuration := "Unit1.Em6.Config".cmMendrelAnodeRearAxisZ,
                           moduleInterface := "Unit1.Em6.HmiInterface".cmMendrelAnodeRearAxisZ,
                           controlNode := "Unit1.Em6.ControlNodes".cmMendrelAnodeRearAxisZ);
END_REGION

REGION Network 176: CmMandrelAnodeRearAxisZ SoftCam
   RUNG wire#powerrail
      "LER_SoftCam_Interface_FC"(actualPosition := "Unit1.Em6.HmiInterface".cmMendrelAnodeRearAxisZ.monitoring.actualPosition, selectSetPosition := "Unit1.Em6.HmiInterface".cmMendrelAnodeRearAxisZ.monitoring.selectSetPosition, softCam := "Unit1.Em6.Config".softCam.cmMendrelAnodeRearAxisZ, position := "Unit1.Em6.Config".cmMendrelAnodeRearAxisZ.setPositions, range := 0.01, softCamPos => "Unit1.Em6.ControlNodes".cm.softCam.mendrelAnodeRearAxisZ)
   END_RUNG
   // the same network as SCL:
   "LER_SoftCam_Interface_FC"(actualPosition := "Unit1.Em6.HmiInterface".cmMendrelAnodeRearAxisZ.monitoring.actualPosition,
                           selectSetPosition := "Unit1.Em6.HmiInterface".cmMendrelAnodeRearAxisZ.monitoring.selectSetPosition,
                           softCam := "Unit1.Em6.Config".softCam.cmMendrelAnodeRearAxisZ,
                           position := "Unit1.Em6.Config".cmMendrelAnodeRearAxisZ.setPositions,
                           range := 0.01,
                           softCamPos => "Unit1.Em6.ControlNodes".cm.softCam.mendrelAnodeRearAxisZ);
END_REGION

REGION Network 178: MendrelCathodeFrontAxisY Enable
   RUNG wire#powerrail
      Contact( "Unit1.EmNodes".sleep.command.Servo.sleep )
      wire#w1
      R_Coil( "Unit1.Em6.ControlNodes".cmMendrelCathodeFrontAxisY.commands.enableAxis )
   END_RUNG
   RUNG wire#powerrail
      Contact( "Unit1.EmNodes".sleep.command.Servo.deppSleep )
   END_RUNG wire#w1
   RUNG wire#powerrail
      Contact( "Unit1.EmNodes".sleep.State.WakeupRecovery )
      S_Coil( "Unit1.Em6.ControlNodes".cmMendrelCathodeFrontAxisY.commands.enableAxis )
   END_RUNG
   // the same network as SCL:
   IF "Unit1.EmNodes".sleep.command.Servo.sleep OR "Unit1.EmNodes".sleep.command.Servo.deppSleep THEN
       "Unit1.Em6.ControlNodes".cmMendrelCathodeFrontAxisY.commands.enableAxis := FALSE;
   END_IF;
   IF "Unit1.EmNodes".sleep.State.WakeupRecovery THEN
       "Unit1.Em6.ControlNodes".cmMendrelCathodeFrontAxisY.commands.enableAxis := TRUE;
   END_IF;
END_REGION

REGION Network 179: CmmendrelCathodeFrontAxisY Home
